# B&R Automation Studio project BottleFiller
Automation Studio 4.11.3.51 SP; technology packages: mapp 5.18.0, mappCockpit 5.18.0, mappMotion 5.18.1, mappView 5.18.1

## Configuration Config1

CPU 5PP5CP.US15-02, AutomationRuntime E4.83, Build 4.1.2, Safety 0.0, Vc V4.72.5

CPU X20CP1586, AutomationRuntime B4.92, Build 4.1.2, Vc V4.72.5

### Task classes (Cpu.sw)
```
Cyclic#4:
  RobVis <- Simulation.Logic.RobVis.prg [disabled]
  BootleFill <- BootleFiller.prg
Libraries: McBase, CoTrace, AsZip, FileIO, runtime, MpUserX, MpBase
```

### Task classes (Cpu.sw)
```
Cyclic#4:
  RobVis <- s.Logic.RobVis.prg
```

### Hardware
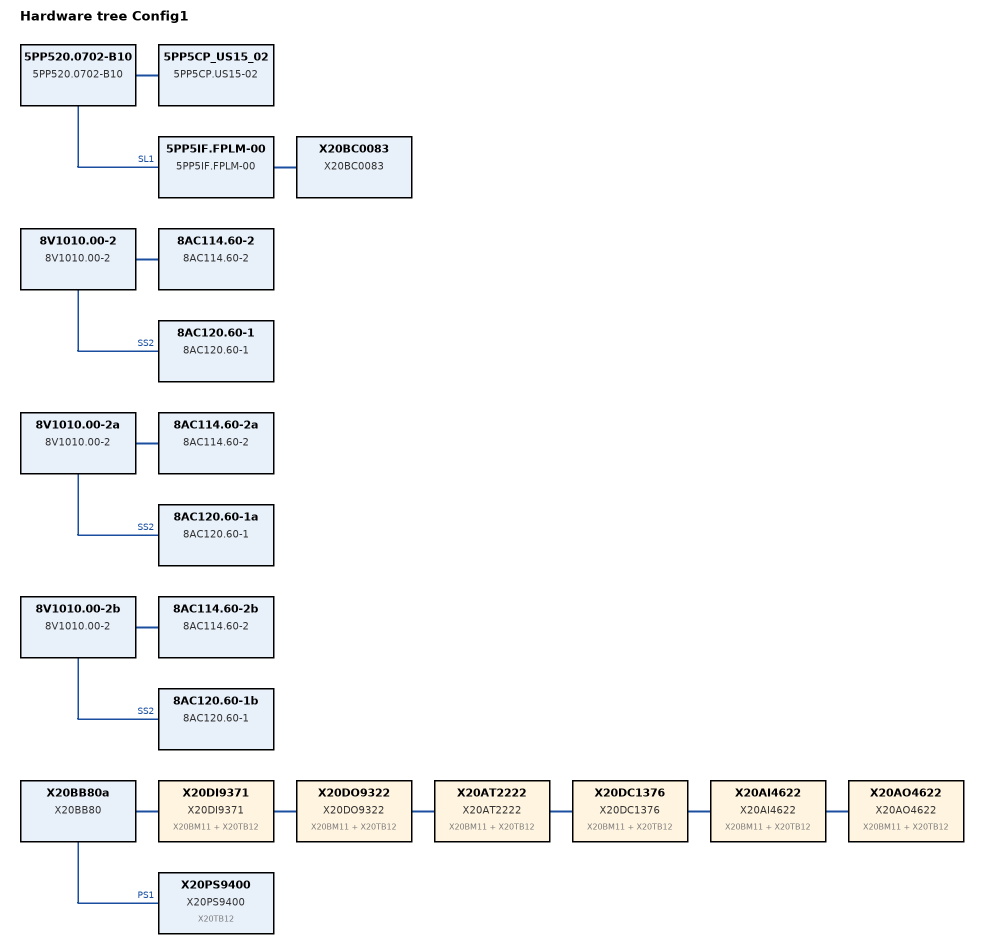
```
5PP520.0702-B10 : 5PP520.0702-B10 v2.0.1.1
  Connector IF3:
    ActivateDevice = 1
    Mode = Manual
    InternetAddress = 192.168.0.121
    SubnetMask = 255.255.255.0
    ActivateSnmp = 2
5PP5CP_US15_02 : 5PP5CP.US15-02 v2.1.6.0  [SY -> 5PP520.0702-B10.SY1]
  ConfigurationID = BottleFiller_Config1
  UserPartitionSize = 10
  FileDevice1
  FileDeviceName1 = USER
  FileDevicePath1 = C:\Recipe\
  ActivateOpcUa = 1
  OpcUaInformationModels_PV_Version = 1
5PP5IF.FPLM-00 : 5PP5IF.FPLM-00 v2.5.0.0  [SL -> 5PP520.0702-B10.SL1]
  Connector IF1:
    Channel1
    ChannelID1 = McAcpBroadcast
8AC114.60-2 : 8AC114.60-2 v1.0.0.8  [SS -> 8V1010.00-2.SS1; PLK1 -> X20BC0083.PLK2 (NodeNumber=2) [Cable Type=PowerlinkCable, Length=10, Version=1.0.0.3]; PLK2 -> 8AC114.60-2a.PLK1 (NodeNumber=2) [Cable Type=PowerlinkCable, Length=10, Version=1.0.0.3]]
8AC114.60-2a : 8AC114.60-2 v1.0.0.8  [SS -> 8V1010.00-2a.SS1; PLK1 -> 8AC114.60-2.PLK2 (NodeNumber=3) [Cable Type=PowerlinkCable, Length=10, Version=1.0.0.3]; PLK2 -> 8AC114.60-2b.PLK1 (NodeNumber=3) [Cable Type=PowerlinkCable, Length=10, Version=1.0.0.3]]
8AC114.60-2b : 8AC114.60-2 v1.0.0.8  [SS -> 8V1010.00-2b.SS1; PLK1 -> 8AC114.60-2a.PLK2 (NodeNumber=4) [Cable Type=PowerlinkCable, Length=10, Version=1.0.0.3]]
8AC120.60-1 : 8AC120.60-1 v2.2.0.0  [SS -> 8V1010.00-2.SS2]
  PlugInType = Encoder
  McAcoposTypeID = AcoposPlugInConfig
8AC120.60-1a : 8AC120.60-1 v2.2.0.0  [SS -> 8V1010.00-2a.SS2]
  PlugInType = Encoder
  McAcoposTypeID = AcoposPlugInConfig
8AC120.60-1b : 8AC120.60-1 v2.2.0.0  [SS -> 8V1010.00-2b.SS2]
  PlugInType = Encoder
  McAcoposTypeID = AcoposPlugInConfig
8V1010.00-2 : 8V1010.00-2 v2.2.0.0
  DriveConfiguration/Module:
    McAcoposTypeID = AcoposConfig
    ActivateACOPOSSimulationOnPLC = 0
    PowerSupply = ETA
  DriveConfiguration/Channel[1]/RealAxis:
    AxisReference = axisConv
    MechanicalElementsIsInvisible = 0
  DriveConfiguration/Channel[1]/RealAxis/MechanicalElements/Gearbox:
    InputIsReadOnly = 0
    Input = 1
    OutputIsReadOnly = 0
    Output = 100
  DriveConfiguration/Channel[1]/RealAxis/MechanicalElements/RotaryToLinearTransformation:
    ReferenceDistanceIsReadOnly = 0
    ReferenceDistance = 1
  DriveConfiguration/Channel[1]/RealAxis/Controller:
    ModeIsReadOnly = 0
    Mode = PositionController
  DriveConfiguration/Channel[1]/RealAxis/Controller/Mode/Position:
    ProportionalGain = 50.0
    IntegrationTime = 0.0
    PredictionTime = 0.0004
    TotalDelayTime = 0.0004
  DriveConfiguration/Channel[1]/RealAxis/Controller/Mode/Speed:
    ProportionalGainIsReadOnly = 0
    ProportionalGain = 2.0
    IntegrationTimeIsReadOnly = 0
    IntegrationTime = 0.0
    FilterTimeIsReadOnly = 0
    FilterTime = 0.0
  DriveConfiguration/Channel[1]/RealAxis/Controller/Mode/LoopFilters:
    LoopFilterXIsReadOnly = 0
    LoopFilter1 = NotUsed
    LoopFilter2 = NotUsed
    LoopFilter3 = NotUsed
  DriveConfiguration/Channel[1]/RealAxis/Homing:
    ModeIsReadOnly = 0
    Mode = Direct
  DriveConfiguration/Channel[1]/RealAxis/Homing/Mode:
    Position = 0.0
    ReferencePulse = NotUsed
  DriveConfiguration/Channel[1]/RealAxis/Homing:
    RestorePositionVariable = 
  DriveConfiguration/Channel[1]/RealAxis/StopReaction:
    QuickstopIsReadOnly = 0
    Quickstop = DecelerationLimit
    DriveErrorIsReadOnly = 0
    DriveError = DecelerationLimit
  DriveConfiguration/Channel[1]/RealAxis/MovementErrorLimits:
    PositionError = 100
    VelocityErrorMonitoring = NotUsed
  DriveConfiguration/Channel[1]/RealAxis:
    JerkFilterIsReadOnly = 0
    JerkFilter = NotUsed
  DriveConfiguration/Channel[1]/RealAxis/DigitalInputs/HomingSwitch:
    SourceIsReadOnly = 0
    Source = X1Ref
    Level = High
  DriveConfiguration/Channel[1]/RealAxis/DigitalInputs/PositiveLimitSwitch:
    Source = X1PosLim
    Level = High
  DriveConfiguration/Channel[1]/RealAxis/DigitalInputs/NegativeLimitSwitch:
    Source = X1NegLim
    Level = High
  DriveConfiguration/Channel[1]/RealAxis/DigitalInputs/Trigger1:
    Source = X1Trigger1
    Level = High
  DriveConfiguration/Channel[1]/RealAxis/DigitalInputs/Trigger2:
    Source = X1Trigger2
    Level = High
  DriveConfiguration/Channel[1]/RealAxis/DigitalInputs/Quickstop:
    Input = Trigger2
  DriveConfiguration/Channel[1]/RealAxis/Simulation:
    SimulationModeOnPLC = SetValueGeneration
    SimulationModeOnACOPOS = NotUsed
  DriveConfiguration/Channel[1]:
    ExternalEncoderAxis = NotUsed
8V1010.00-2a : 8V1010.00-2 v2.2.0.0
  DriveConfiguration/Module:
    McAcoposTypeID = AcoposConfig
    ActivateACOPOSSimulationOnPLC = 1
    PowerSupply = ETA
  DriveConfiguration/Channel[1]/RealAxis:
    AxisReference = axisCart
    MechanicalElementsIsInvisible = 0
  DriveConfiguration/Channel[1]/RealAxis/MechanicalElements/Gearbox:
    InputIsReadOnly = 0
    Input = 1
    OutputIsReadOnly = 0
    Output = 1
  DriveConfiguration/Channel[1]/RealAxis/MechanicalElements/RotaryToLinearTransformation:
    ReferenceDistanceIsReadOnly = 0
    ReferenceDistance = 1
  DriveConfiguration/Channel[1]/RealAxis/Controller:
    ModeIsReadOnly = 0
    Mode = PositionController
  DriveConfiguration/Channel[1]/RealAxis/Controller/Mode/Position:
    ProportionalGain = 50.0
    IntegrationTime = 0.0
    PredictionTime = 0.0004
    TotalDelayTime = 0.0004
  DriveConfiguration/Channel[1]/RealAxis/Controller/Mode/Speed:
    ProportionalGainIsReadOnly = 0
    ProportionalGain = 2.0
    IntegrationTimeIsReadOnly = 0
    IntegrationTime = 0.0
    FilterTimeIsReadOnly = 0
    FilterTime = 0.0
  DriveConfiguration/Channel[1]/RealAxis/Controller/Mode/LoopFilters:
    LoopFilterXIsReadOnly = 0
    LoopFilter1 = NotUsed
    LoopFilter2 = NotUsed
    LoopFilter3 = NotUsed
  DriveConfiguration/Channel[1]/RealAxis/Homing:
    ModeIsReadOnly = 0
    Mode = Direct
  DriveConfiguration/Channel[1]/RealAxis/Homing/Mode:
    Position = 0.0
    ReferencePulse = NotUsed
  DriveConfiguration/Channel[1]/RealAxis/Homing:
    RestorePositionVariable = 
  DriveConfiguration/Channel[1]/RealAxis/StopReaction:
    QuickstopIsReadOnly = 0
    Quickstop = DecelerationLimit
    DriveErrorIsReadOnly = 0
    DriveError = DecelerationLimit
  DriveConfiguration/Channel[1]/RealAxis/MovementErrorLimits:
    PositionError = 1.0
    VelocityErrorMonitoring = Automatic1
  DriveConfiguration/Channel[1]/RealAxis:
    JerkFilterIsReadOnly = 0
    JerkFilter = NotUsed
  DriveConfiguration/Channel[1]/RealAxis/DigitalInputs/HomingSwitch:
    SourceIsReadOnly = 0
    Source = X1Ref
    Level = High
  DriveConfiguration/Channel[1]/RealAxis/DigitalInputs/PositiveLimitSwitch:
    Source = X1PosLim
    Level = High
  DriveConfiguration/Channel[1]/RealAxis/DigitalInputs/NegativeLimitSwitch:
    Source = X1NegLim
    Level = High
  DriveConfiguration/Channel[1]/RealAxis/DigitalInputs/Trigger1:
    Source = X1Trigger1
    Level = High
  DriveConfiguration/Channel[1]/RealAxis/DigitalInputs/Trigger2:
    Source = X1Trigger2
    Level = High
  DriveConfiguration/Channel[1]/RealAxis/DigitalInputs/Quickstop:
    Input = Trigger2
  DriveConfiguration/Channel[1]/RealAxis/Simulation:
    SimulationModeOnPLC = SetValueGeneration
    SimulationModeOnACOPOS = CompleteControlledSystem
  DriveConfiguration/Channel[1]/RealAxis/Simulation/SimulationModeOnACOPOS:
    LoadModel = OneMassBasedOnMotorParameters
  DriveConfiguration/Channel[1]/RealAxis/Simulation/SimulationModeOnACOPOS/LoadModel:
    AdditiveLoadParID = 0
  DriveConfiguration/Channel[1]/RealAxis/AxisFeatures:
    FeatureRef[1] = Feature_CamAutomat
  DriveConfiguration/Channel[1]:
    ExternalEncoderAxis = NotUsed
8V1010.00-2b : 8V1010.00-2 v2.2.0.0
  DriveConfiguration/Module:
    McAcoposTypeID = AcoposConfig
    ActivateACOPOSSimulationOnPLC = 1
    PowerSupply = ETA
  DriveConfiguration/Channel[1]/RealAxis:
    AxisReference = axisNozzle
    MechanicalElementsIsInvisible = 0
  DriveConfiguration/Channel[1]/RealAxis/MechanicalElements/Gearbox:
    InputIsReadOnly = 0
    Input = 1
    OutputIsReadOnly = 0
    Output = 1
  DriveConfiguration/Channel[1]/RealAxis/MechanicalElements/RotaryToLinearTransformation:
    ReferenceDistanceIsReadOnly = 0
    ReferenceDistance = 1
  DriveConfiguration/Channel[1]/RealAxis/Controller:
    ModeIsReadOnly = 0
    Mode = PositionController
  DriveConfiguration/Channel[1]/RealAxis/Controller/Mode/Position:
    ProportionalGain = 2
    IntegrationTime = 0.0
    PredictionTime = 0.0004
    TotalDelayTime = 0.0004
  DriveConfiguration/Channel[1]/RealAxis/Controller/Mode/Speed:
    ProportionalGainIsReadOnly = 0
    ProportionalGain = 0.01
    IntegrationTimeIsReadOnly = 0
    IntegrationTime = 0.0
    FilterTimeIsReadOnly = 0
    FilterTime = 0.0
  DriveConfiguration/Channel[1]/RealAxis/Controller/Mode/LoopFilters:
    LoopFilterXIsReadOnly = 0
    LoopFilter1 = NotUsed
    LoopFilter2 = NotUsed
    LoopFilter3 = NotUsed
  DriveConfiguration/Channel[1]/RealAxis/Homing:
    ModeIsReadOnly = 0
    Mode = Direct
  DriveConfiguration/Channel[1]/RealAxis/Homing/Mode:
    Position = 195.0
    ReferencePulse = NotUsed
  DriveConfiguration/Channel[1]/RealAxis/Homing:
    RestorePositionVariable = 
  DriveConfiguration/Channel[1]/RealAxis/StopReaction:
    QuickstopIsReadOnly = 0
    Quickstop = DecelerationLimit
    DriveErrorIsReadOnly = 0
    DriveError = DecelerationLimit
  DriveConfiguration/Channel[1]/RealAxis/MovementErrorLimits:
    PositionError = 1.0
    VelocityErrorMonitoring = Automatic1
  DriveConfiguration/Channel[1]/RealAxis:
    JerkFilterIsReadOnly = 0
    JerkFilter = NotUsed
  DriveConfiguration/Channel[1]/RealAxis/DigitalInputs/HomingSwitch:
    SourceIsReadOnly = 0
    Source = X1Ref
    Level = High
  DriveConfiguration/Channel[1]/RealAxis/DigitalInputs/PositiveLimitSwitch:
    Source = X1PosLim
    Level = High
  DriveConfiguration/Channel[1]/RealAxis/DigitalInputs/NegativeLimitSwitch:
    Source = X1NegLim
    Level = High
  DriveConfiguration/Channel[1]/RealAxis/DigitalInputs/Trigger1:
    Source = X1Trigger1
    Level = High
  DriveConfiguration/Channel[1]/RealAxis/DigitalInputs/Trigger2:
    Source = X1Trigger2
    Level = High
  DriveConfiguration/Channel[1]/RealAxis/DigitalInputs/Quickstop:
    Input = Trigger2
  DriveConfiguration/Channel[1]/RealAxis/Simulation:
    SimulationModeOnPLC = SetValueGeneration
    SimulationModeOnACOPOS = NotUsed
  DriveConfiguration/Channel[1]/RealAxis/AxisFeatures:
    FeatureRef[1] = Feature_CamList
  DriveConfiguration/Channel[1]:
    ExternalEncoderAxis = NotUsed
  DriveConfiguration/Channel[1]/ChannelFeatures:
    FeatureRef[1] = Feature_CamList_1
X20AI4622 : X20AI4622 v1.2.0.0  [SS1 -> X20TB12f.SS; SL -> X20BM11e.SL1]
X20AO4622 : X20AO4622 v1.3.0.0  [SS1 -> X20TB12g.SS; SL -> X20BM11f.SL1]
X20AT2222 : X20AT2222 v1.4.0.0  [SS1 -> X20TB12d.SS; SL -> X20BM11c.SL1]
X20BB80a : X20BB80 v1.1.0.0
X20BC0083 : X20BC0083 v2.12.0.0  [PLK1 -> 5PP5IF.FPLM-00.IF1 (NodeNumber=1) [Cable Type=PowerlinkCable, Length=10, Version=1.0.0.3]; PLK2 -> 8AC114.60-2.PLK1 (NodeNumber=1) [Cable Type=PowerlinkCable, Length=10, Version=1.0.0.3]; SL -> X20BB80a.SL1]
  Supervision = off
X20BM11a : X20BM11 v1.1.0.0  [X2X1 -> X20BB80a.IF1]
X20BM11b : X20BM11 v1.1.0.0  [X2X1 -> X20BM11a.X2X2]
X20BM11c : X20BM11 v1.1.0.0  [X2X1 -> X20BM11b.X2X2]
X20BM11d : X20BM11 v1.1.0.0  [X2X1 -> X20BM11c.X2X2]
X20BM11e : X20BM11 v1.1.0.0  [X2X1 -> X20BM11d.X2X2]
X20BM11f : X20BM11 v1.1.0.0  [X2X1 -> X20BM11e.X2X2]
X20DC1376 : X20DC1376 v1.3.0.0  [SS1 -> X20TB12e.SS; SL -> X20BM11d.SL1]
X20DI9371 : X20DI9371 v1.3.0.0  [SS1 -> X20TB12a.SS; SL -> X20BM11a.SL1]
X20DO9322 : X20DO9322 v1.4.0.0  [SS1 -> X20TB12c.SS; SL -> X20BM11b.SL1]
X20PS9400 : X20PS9400 v1.7.0.0  [SS1 -> X20TB12b.SS; PS -> X20BB80a.PS1]
  Supervision = off
X20TB12a : X20TB12 v1.0.0.0
X20TB12b : X20TB12 v1.0.0.0
X20TB12c : X20TB12 v1.0.0.0
X20TB12d : X20TB12 v1.0.0.0
X20TB12e : X20TB12 v1.0.0.0
X20TB12f : X20TB12 v1.0.0.0
X20TB12g : X20TB12 v1.0.0.0
```

### Config_1.axis - 5PP5CP_US15_02/mappMotion/Config_1.axis
```
Element axisConv (Type=axis)
  BaseTypeIsReadOnly = 0
  BaseType = LinearPeriodic
    MeasurementUnit = 5066068
    MeasurementResolutionIsReadOnly = 0
    MeasurementResolution = 0.01
    CountDirectionIsReadOnly = 0
    CountDirection = Standard
    PeriodSettings:
      Period = 5000
  MovementLimitsIsReadOnly = 0
  MovementLimits = Internal
    Position:
      LowerLimitMin = -1.79769313486231E308
      UpperLimitMax = 1.79769313486231E308
      LowerLimit = -1000.0
      UpperLimit = 1000.0
    VelocityIsReadOnly = 0
    Velocity:
      VelocityMax = 3.4E38
      Velocity = 10.0
    AccelerationIsReadOnly = 0
    Acceleration:
      AccelerationMax = 3.4E38
      Acceleration = 50.0
    DecelerationIsReadOnly = 0
    Deceleration:
      DecelerationMax = 3.4E38
      Deceleration = 50.0
  Alarms = None
Element axisCart (Type=axis)
  BaseTypeIsReadOnly = 0
  BaseType = LinearPeriodic
    MeasurementUnit = 5066068
    MeasurementResolutionIsReadOnly = 0
    MeasurementResolution = 0.01
    CountDirectionIsReadOnly = 0
    CountDirection = Standard
    PeriodSettings:
      Period = 1200
  MovementLimitsIsReadOnly = 0
  MovementLimits = Internal
    Position:
      LowerLimitMin = -1.79769313486231E308
      UpperLimitMax = 1.79769313486231E308
      LowerLimit = -1000.0
      UpperLimit = 1000.0
    VelocityIsReadOnly = 0
    Velocity:
      VelocityMax = 3.4E38
      Velocity = 10.0
    AccelerationIsReadOnly = 0
    Acceleration:
      AccelerationMax = 3.4E38
      Acceleration = 50.0
    DecelerationIsReadOnly = 0
    Deceleration:
      DecelerationMax = 3.4E38
      Deceleration = 50.0
  Alarms = None
Element axisNozzle (Type=axis)
  BaseTypeIsReadOnly = 0
  BaseType = LinearPeriodic
    MeasurementUnit = 5066068
    MeasurementResolutionIsReadOnly = 0
    MeasurementResolution = 0.01
    CountDirectionIsReadOnly = 0
    CountDirection = Standard
    PeriodSettings:
      Period = 200
  MovementLimitsIsReadOnly = 0
  MovementLimits = Internal
    Position:
      LowerLimitMin = -1.79769313486231E308
      UpperLimitMax = 1.79769313486231E308
      LowerLimit = -1000.0
      UpperLimit = 1000.0
    VelocityIsReadOnly = 0
    Velocity:
      VelocityMax = 3.4E38
      Velocity = 10.0
    AccelerationIsReadOnly = 0
    Acceleration:
      AccelerationMax = 3.4E38
      Acceleration = 50.0
    DecelerationIsReadOnly = 0
    Deceleration:
      DecelerationMax = 3.4E38
      Deceleration = 50.0
  Alarms = None
```

### Config_1.camlist - 5PP5CP_US15_02/mappMotion/Config_1.camlist
```
Element CamList_1 (Type=camlist)
  Row[1]:
    CamName = b1_Nozzle
    CamID = 1
    Description
```

### Config_2.axisfeature - 5PP5CP_US15_02/mappMotion/Config_2.axisfeature
```
Element Feature_CamList_1 (Type=axisfeature)
  Type = CamList
    CamListRef = CamList_1
```

### configAxis.axis - 5PP5CP_US15_02/mappMotion/configAxis.axis
```
Element axisConv (Type=axis)
  BaseTypeIsReadOnly = 0
  BaseType = LinearPeriodic
    MeasurementUnit = 5066068
    MeasurementResolutionIsReadOnly = 0
    MeasurementResolution = 0.01
    CountDirectionIsReadOnly = 0
    CountDirection = Standard
    PeriodSettings:
      Period = 5000
  MovementLimitsIsReadOnly = 0
  MovementLimits = Internal
    Position:
      LowerLimitMin = -1.79769313486231E308
      UpperLimitMax = 1.79769313486231E308
      LowerLimit = -1000.0
      UpperLimit = 1000.0
    VelocityIsReadOnly = 0
    Velocity:
      VelocityMax = 3.4E38
      Velocity = 600
    AccelerationIsReadOnly = 0
    Acceleration:
      AccelerationMax = 3.4E38
      Acceleration = 10000
    DecelerationIsReadOnly = 0
    Deceleration:
      DecelerationMax = 3.4E38
      Deceleration = 100000
  Alarms = MpAlarmX
    mapp.AlarmX.Core.Configuration:
      [0]:
        Message = Conveyor system problem
        Code = 100
        Severity = 10
      [3]:
        Message = Conveyor Operation Problem
        Code = 200
        Severity = 20
      [14]:
        Message = Conveyor Motor problem
        Code = 300
        Severity = 30
Element axisCart (Type=axis)
  BaseTypeIsReadOnly = 0
  BaseType = LinearBounded
    MeasurementUnit = 5066068
    MeasurementResolutionIsReadOnly = 0
    MeasurementResolution = 0.01
    CountDirectionIsReadOnly = 0
    CountDirection = Standard
  MovementLimitsIsReadOnly = 0
  MovementLimits = Internal
    Position:
      LowerLimitMin = -1.79769313486231E308
      UpperLimitMax = 1.79769313486231E308
      LowerLimit = -100
      UpperLimit = 1100
    VelocityIsReadOnly = 0
    Velocity:
      VelocityMax = 3.4E38
      Velocity = 800
    AccelerationIsReadOnly = 0
    Acceleration:
      AccelerationMax = 3.4E38
      Acceleration = 10000
    DecelerationIsReadOnly = 0
    Deceleration:
      DecelerationMax = 3.4E38
      Deceleration = 100000
  Alarms = MpAlarmX
    mapp.AlarmX.Core.Configuration:
      [0]:
        Message = Cart System problem
        Code = 101
        Severity = 10
      [3]:
        Message = Cart Operation problem
        Code = 201
        Severity = 20
      [14]:
        Message = Cart Motor problem
        Code = 301
        Severity = 30
Element axisNozzle (Type=axis)
  BaseTypeIsReadOnly = 0
  BaseType = LinearBounded
    MeasurementUnit = 5066068
    MeasurementResolutionIsReadOnly = 0
    MeasurementResolution = 0.01
    CountDirectionIsReadOnly = 0
    CountDirection = Standard
  MovementLimitsIsReadOnly = 0
  MovementLimits = Internal
    Position:
      LowerLimitMin = -1.79769313486231E308
      UpperLimitMax = 1.79769313486231E308
      LowerLimit = 0
      UpperLimit = 200
    VelocityIsReadOnly = 0
    Velocity:
      VelocityMax = 3.4E38
      Velocity = 5000
    AccelerationIsReadOnly = 0
    Acceleration:
      AccelerationMax = 3.4E38
      Acceleration = 20000
    DecelerationIsReadOnly = 0
    Deceleration:
      DecelerationMax = 3.4E38
      Deceleration = 800000
  Alarms = MpAlarmX
    mapp.AlarmX.Core.Configuration:
      [0]:
        Message = Nozzle System problem
        Code = 102
        Severity = 10
      [3]:
        Message = Nozzle Operation problem
        Code = 202
        Severity = 20
      [14]:
        Message = Nozzle Motor problem
        Code = 302
        Severity = 30
```

### configCam.axisfeature - 5PP5CP_US15_02/mappMotion/configCam.axisfeature
```
Element Feature_CamAutomat (Type=axisfeature)
  Type = CamAutomat
    CamAutomatType = ACOPOS
      CommonParameters:
        Master:
          ValueSource = SetPosition
            AxisReference
            MaxVelocity = 1.0
          StartPosition = 0.0
          StartInterval = MasterAxisPeriod
        AdvancedParameters:
          StartStateParameters:
            StartState = 0
            RelMasterStartPos = 0.0
          AdditiveAxes:
            AdditiveMasterValueSource = NotUsed
            AdditiveSlaveValueSource = NotUsed
          MasterStartPositionMode = NotEvaluatedAnew
          ControlSettings:
            CrossLeftBoundary = PositionLimitedHorizontal
            CamChangeImmediately = CurrentMasterMoveDir
          MessageSettings:
            ErrorsInStandby = NoErrorMessages
          TriggerAndLatch:
            Trigger1Delay = 0.0
            Trigger2Delay = 0.0
            SlaveLatchParID = 0
          EventParIDs
          StartIntervals
          Factors:
            SlaveFactorParID = 0
      States:
        State0 = Used
```

### configNozz.axisfeature - 5PP5CP_US15_02/mappMotion/configNozz.axisfeature
```
Element Feature_CamList (Type=axisfeature)
  Type = CamAutomat
    CamAutomatType = ACOPOS
      CommonParameters:
        Master:
          ValueSource = SetPosition
            AxisReference = axisConv
            MaxVelocity = 600
          StartPosition = 0.0
          StartInterval = MasterAxisPeriod
        AdvancedParameters:
          StartStateParameters:
            StartState = 0
            RelMasterStartPos = 0.0
          AdditiveAxes:
            AdditiveMasterValueSource = NotUsed
            AdditiveSlaveValueSource = NotUsed
          MasterStartPositionMode = NotEvaluatedAnew
          ControlSettings:
            CrossLeftBoundary = PositionLimitedHorizontal
            CamChangeImmediately = CurrentMasterMoveDir
          MessageSettings:
            ErrorsInStandby = NoErrorMessages
          TriggerAndLatch:
            Trigger1Delay = 0.0
            Trigger2Delay = 0.0
            SlaveLatchParID = 0
          EventParIDs
          StartIntervals
          Factors:
            SlaveFactorParID = 0
      States:
        State0 = Used
          Events:
            Event[0]:
              Type = Signal1FromPLC
              Transition = Immediately
              SynchronousUpdate = Used
              NextState = 1
        State[1]:
          Cam = Predefined
            PredefinedCam = ZeroPoint
          MasterFactor = 100
          SlaveFactor = -100
          CompensationMode = MasterSlaveAbsolutePosition
            MasterPosition = 90
            SlavePosition = 195
            MaxSlaveVelocity = 1000
            MaxSlaveAcceleration1 = 2000
            MaxSlaveAcceleration2 = 2250
            AdvancedParameters = NotUsed
          AdvancedParameters:
            RepeatCounterInit = 0
            MasterValueSource = CommonMaster
          Events:
            Event[0]:
              Type = StateEnd
              Transition = EndOfState
              SynchronousUpdate = NotUsed
              NextState = 2
        State[2]:
          Cam = Predefined
            PredefinedCam = OneToOne
          MasterFactor = 100
          SlaveFactor = 100
          CompensationMode = SlaveCompensationAbsSlPos
            MasterDistance = 50
            SlavePosition = 5
            AdvancedParameters = NotUsed
          AdvancedParameters:
            RepeatCounterInit = 0
            MasterValueSource = CommonMaster
          Events:
            Event[0]:
              Type = StateEnd
              Transition = EndOfState
              SynchronousUpdate = NotUsed
              NextState = 3
        State[3]:
          Cam = CamID
            CamID = 1
          MasterFactor = 40000
          SlaveFactor = 19000
          CompensationMode = NoCompensation
          AdvancedParameters:
            RepeatCounterInit = 0
            MasterValueSource = CommonMaster
          Events:
            Event[0]:
              Type = StateEnd
              Transition = EndOfState
              SynchronousUpdate = NotUsed
              NextState = 4
        State[4]:
          Cam = Predefined
            PredefinedCam = ZeroPoint
          MasterFactor = 100
          SlaveFactor = 100
          CompensationMode = SlaveCompensationAbsSlPos
            MasterDistance = 50
            SlavePosition = 195
            AdvancedParameters = NotUsed
          AdvancedParameters:
            RepeatCounterInit = 0
            MasterValueSource = CommonMaster
          Events:
            Event[0]:
              Type = StateEnd
              Transition = Immediately
              SynchronousUpdate = NotUsed
              NextState = 2
```

### alarm.mpalarmxcore - 5PP5CP_US15_02/mappServices/alarm.mpalarmxcore
```
Element gBFAlarmXCore (Type=mpalarmxcore)
  mapp.AlarmX.Core.Configuration:
    [0]:
      Name = noPower
      Message = You should click PowerSwitch first.
      Code = 99
      Severity = 10
      Behavior = PersistentAlarm
```

### fileM.mpfilemanager - 5PP5CP_US15_02/mappServices/fileM.mpfilemanager
```
Element FileManagement (Type=mpfilemanager)
  FileManager:
    Devices:
      0:
        DeviceName = USER
        Text = Recipe
    Access:
      0:
        Folder = *
        Roles:
          0:
            Role = Shift Leader
            Rights:
              Visible = TRUE
              FolderRead = TRUE
              FileRead = TRUE
              FileEdit = TRUE
              FolderEdit = TRUE
    Auditing = MpAudit
      Read = TRUE
  FileManagerRestrict:
    0:
      0:
        Folder = 
    1:
      Functionality = TextEditor
      0:
        Folder = C:\Recipe
        Restrictions:
          BrowseUp = TRUE
          BrowseDown = TRUE
          ReadOnly = TRUE
          CreatFolders = TRUE
```

### recipeXML.mprecipexml - 5PP5CP_US15_02/mappServices/recipeXML.mprecipexml
```
Element BFRecipe (Type=mprecipexml)
  mapp.Recipe.Xml:
    Auditing = MpAudit
```

## Logical view

Binary libraries used (declarations not repeated): operator, runtime, astime, AsIecCon, McBase, CoTrace, AsZip, FileIO, MpUserX, MpBase

### Global.var - Global variables
```iecst
VAR
	roleInfo : MpUserXMgrUIRoleInfoType;
	role : MpUserXMgrUIUserInfoType;
END_VAR
```

### Package Logical/Libraries - Global libraries

### BF_GlobarVar.var
```iecst
VAR
	gFillerTyp : gBFWorkEnum;
	gAxisCase : gBFCaseEnum;
	gControl : gManagementTyp;
	gAxisUpdate : gAxisUpdateParType;
	gMainAction : gMainActionTyp;
	gAxisOutputs : gAxisOutputsTyp;
	gCamSeqParam : camSequencersParams;
	gCaseError : gErrorCaseEnum;
	gMain : gFillerEnum;
	gPump : gPumpMgmtTyp;
	temp : BOOL := FALSE;
END_VAR
```

### BF_GlobalTyp.typ
```iecst
TYPE
	gPumpMgmtTyp : 	STRUCT
		PumpFlowSpeed : USINT;
		PumpRelay : USINT := 0;
		ValveStatus : STRING[80];
		ValveRelay : BOOL := FALSE;
	END_STRUCT;
	camSequencersParams : 	STRUCT
		cart : camParam; (*Parametry cama karetki*)
		nozzle : camParam; (*Parametry cama dysz*)
	END_STRUCT;
	camParam : 	STRUCT
		signal1 : BOOL := FALSE; (*Wyzwalanie signal1*)
		currentStateIndex : INT := 0; (*Zwraca aktualny state*)
	END_STRUCT;
	gAxisOutputsTyp : 	STRUCT
		Conveyor : gControlInfoTyp;
		Cart : gControlInfoTyp;
		Nozzle : gControlInfoTyp;
		currentBottleType : UINT := 1; (*Aktualny typ butelki*)
		velocity : REAL; (*Aktualna prędkość*)
	END_STRUCT;
	gControlInfoTyp : 	STRUCT  (*parameters, output*)
		error : BOOL := FALSE; (*error*)
		isPowered : BOOL := FALSE; (*jest zasilony*)
		isHomed : BOOL := FALSE; (*jest w pozycji home*)
		position : REAL := 0; (*aktualna pozycja*)
		velocity : REAL := 0; (*aktualne velocity*)
		updateDone : BOOL := FALSE;
		MoveActive : BOOL := FALSE;
		Direction : STRING[80];
	END_STRUCT;
	gControlTyp : 	STRUCT  (*parameters, inputs*)
		power : BOOL := FALSE; (*Uruchomienie maszyny*)
		errorReset : BOOL := FALSE;
		autoTune : BOOL := TRUE;
		home : BOOL := FALSE;
		jogNegative : BOOL := FALSE;
		jogPositive : BOOL := FALSE;
		moveVelocity : BOOL := FALSE;
		stop : BOOL := FALSE;
		currentBottleType : STRING[80] := '1';
		safeLevelStop : BOOL; (*Informuje, czy w trybie półautomatycznym przekroczone zostały bezpieczne granice*)
		onlyLeft : BOOL := FALSE; (*Wskazuje, że w trybie półautomatycznym możliwy aktualnie jest ruch tylko w lewo*)
		onlyRight : BOOL := FALSE; (*Wskazuje, że w trybie półautomatycznym możliwy aktualnie jest ruch tylko w prawo*)
		upperLimit : INT; (*Maksymalne velocity Operatora*)
		lowerLimit : INT; (*Minimalne velocity Operatora*)
		Direction : STRING[80];
	END_STRUCT;
	gMainActionTyp : 	STRUCT  (*Flagi pomocne w sterowaniu projektem*)
		powered : BOOL := FALSE; (*Czy maszyna jest zasilona*)
		homed : BOOL := FALSE; (*Czy maszyna jest home'owana*)
		connected : BOOL := FALSE; (*Czy osie są połączone*)
		disconnected : BOOL := FALSE; (*Czy osie są rozłączone*)
		stopped : BOOL := FALSE; (*Czy Osie stoją*)
	END_STRUCT;
	gAxisUpdateParType : 	STRUCT  (*update parameters structure*)
		Conveyor : gParametersUpdate;
		Cart : gParametersUpdate;
		Nozzle : gParametersUpdate;
		staticVelocity : STRING[80] := '10'; (*Static velocity to veloocity z opcji "Slow", "Normal", "Fast"*)
	END_STRUCT;
	gManagementTyp : 	STRUCT  (*Zarządzanie maszyną*)
		Conveyor : gControlTyp;
		Cart : gControlTyp;
		Nozzle : gControlTyp;
		power : BOOL := FALSE; (*Zasilenie maszyny*)
		start : BOOL := FALSE; (*Start maszyny*)
		stop : BOOL := FALSE; (*Stop maszyny*)
		manual : BOOL := FALSE; (*Manualna praca*)
		inCam : BOOL := FALSE; (*Flaga wskazująca na status połączenia osi*)
		needUpdate : BOOL := TRUE; (*Flaga wskazująca na konieczność aktualizacji*)
		moveVelocity : BOOL := FALSE; (*Wyzwolenie ruchu*)
		disconnect : BOOL := FALSE; (*Rozłączenie osi*)
		bottleCnt : INT := 0; (*Liczy butelki*)
		currentBottleType : STRING[80] := '1'; (*Aktualny typ butelki*)
		part : REAL; (*5% z aktualnej prędkości*)
		partVelUpd : BOOL := FALSE; (*Flaga wskazująca na konieczność aktualizacji prędkości*)
		maxVelocity : REAL; (*Maksymalne Velocity Operatora*)
		decVisible : BOOL := TRUE; (*Widoczność przycisku Decrease*)
		emergencySTOP : BOOL := FALSE;
		switchToAutomat : BOOL := FALSE;
		incVisible : BOOL := TRUE; (*Widoczność przycisku Increase*)
		minVelocity : REAL; (*Minimalne Velocity Operatora*)
		startSeq : BOOL := TRUE;
	END_STRUCT;
	gErrorCaseEnum :
		(
		noError,
		handleError,
		inError
		);
	gFillerEnum :
		( (*Every possible case*)
		DISABLED,
		INIT,
		WORK,
		STOP,
		ERROR
		);
	gParametersUpdate : 	STRUCT  (*update parameters*)
		Velocity : REAL := 10;
		Direction : REAL := 1;
		FirstPosition : REAL := 0;
		LastPosition : REAL := 0;
		Position : REAL := 0;
		Homing : REAL := 0;
	END_STRUCT;
	gBFWorkEnum :
		( (*BF_Work control*)
		WAITING, (*Stan początkowy*)
		AUTOMAT, (*Tryb automatyczny*)
		MANUAL (*Tryb manualny*)
		);
	gBFCaseEnum :
		( (*BF_Axis control*)
		WAIT, (*Tryb początkowy*)
		STANDSTILL, (*Czeka na ruch*)
		POWERED, (*Maszyna zasilona*)
		HOLDON, (*Zatrzymanie maszyny*)
		CONNECT, (*Połączenie osi*)
		onMOVE, (*W ruchu*)
		DISCONNECT, (*Rozłączenie osi*)
		HOMING (*Przywrócenie pozycji początkowych*)
		);
END_TYPE
```

### Program Logical/BottleFiller/BF_Main (IEC)

#### Types.typ
```iecst
TYPE
	SimulationAxisPositionEnum : 	STRUCT
		Conveyor : REAL;
		Cart : REAL;
		Nozzle : REAL;
	END_STRUCT;
	bottleFillerRecipeEnum : 	STRUCT
		diPumpSpeedFlow : INT := 0;
		diVelocity : REAL := 0.0;
		diSpeedProfile : INT := 0;
		diBottleShape : INT := 0;
	END_STRUCT;
END_TYPE
```

#### Variables.var
```iecst
(*case machine*)
VAR
	bottleFillerRecipeTyp : bottleFillerRecipeEnum;
END_VAR
(*digital inputs*)
VAR
	diError : BOOL;
	diManual : BOOL := FALSE; (*Determine if machine works automatically or needs manual control*)
	diStop : BOOL := FALSE; (*Stop switch*)
	diStart : BOOL := FALSE; (*Start switch*)
	diPowerSwitch : BOOL := FALSE; (*Power on switch*)
	diLiquidLevel : REAL := 100;
	diConveyorHomingSwitch : BOOL := FALSE; (*Sensor detecting conveyor at homing position*)
	diNozzleHomingSwitch : BOOL := FALSE; (*Sensor detecting nozzle at homing position*)
	diCartHomingSwitch : BOOL := FALSE; (*Sensor detecting cart at homing position*)
	diBottleDetection : BOOL := FALSE; (*Sensor detecting presence of a bottle*)
END_VAR
(*digital outputs*)
VAR
	doPumpRelay : INT; (*Output controlling the pump building pressure for liquid flow*)
	doValveRelay : BOOL; (*Output controlling the liquid valve opening*)
END_VAR
(*analog outputs*)
VAR
	aoPumpFlowSpeed : ARRAY[0..100] OF INT; (*Datapoint in percentage to the pump system about liquid flow speed in percent*)
END_VAR
(*other variables*)
VAR
	result : INT;
	counter : INT;
	roleInfo : MpUserXMgrUIRoleInfoType;
	MpBFRecipeXml : MpRecipeXml;
	MpBFRecipeRegPar : MpRecipeRegPar; (*MpBFRecipeHMI : MpRecipeUI;
	UISetup : MpRecipeUISetupType;
	MpRecipeUIConnectType : MpRecipeUIConnectType;*)
	inCam : BOOL;
	SimulationAxisPosition : SimulationAxisPositionEnum;
	changedPosition : BOOL;
END_VAR
```

#### Main.st
```iecst
PROGRAM _INIT
	(* Insert code here *)
	 gMain:=DISABLED;
END_PROGRAM

PROGRAM _CYCLIC
	(* Insert code here *)

	SimulationAxisPosition.Cart := LREAL_TO_REAL(gAxisOutputs.Cart.position);
	SimulationAxisPosition.Conveyor := LREAL_TO_REAL(gAxisOutputs.Conveyor.position);
	SimulationAxisPosition.Nozzle := LREAL_TO_REAL(gAxisOutputs.Nozzle.position);
	gAdrAxesPositions := ADR(SimulationAxisPosition);

	CASE gMain OF
		DISABLED:
			diStart:=0;
			diStop:=0;

			IF gControl.power THEN
				gMain:=INIT;
			END_IF;

		INIT:
			gControl.Cart.lowerLimit:=-95;
			gControl.Cart.upperLimit:=1095;

			gControl.Conveyor.lowerLimit:=0;
			gControl.Conveyor.upperLimit:=4997;

			gControl.Nozzle.lowerLimit:=2;
			gControl.Nozzle.upperLimit:=197;

			gAxisCase:=POWERED;

			IF gMainAction.powered AND NOT gControl.inCam THEN
				gAxisCase:=HOMING;
			END_IF;

			IF gMainAction.powered AND gMainAction.homed THEN
				gControl.Cart.home:=0;
				gControl.Conveyor.home:=0;
				gControl.Nozzle.home:=0;
				gAxisCase:=STANDSTILL;
			END_IF;

			IF gMainAction.powered AND gMainAction.homed AND gControl.start AND NOT gControl.manual THEN
				gAxisCase:=CONNECT;
				IF gMainAction.connected THEN
					gAxisCase:=onMOVE;
					gFillerTyp:=AUTOMAT;
					gMain:=WORK;
				END_IF;
			END_IF;

			IF gMainAction.powered AND gMainAction.homed AND gControl.start AND gControl.manual THEN
				gMainAction.homed:=0;
				gAxisCase:=onMOVE;
				gFillerTyp:=MANUAL;
				gMain:=WORK;
			END_IF;

		WORK:
			result:= gControl.bottleCnt MOD 5;

			IF result=1 THEN
				gCamSeqParam.nozzle.signal1:=1;
			END_IF;
			IF result <> 1 THEN
				gCamSeqParam.nozzle.signal1:=0;
				gCamSeqParam.cart.signal1:=0;
			END_IF;

			IF (gCamSeqParam.nozzle.currentStateIndex = 3) AND (gAxisOutputs.Nozzle.position > 0 AND gAxisOutputs.Nozzle.position < 170) THEN
				gPump.ValveRelay:=1;
				gPump.ValveStatus:='Opened';
			ELSE
				gPump.ValveRelay:=0;
				gPump.ValveStatus:='Closed';
			END_IF;

		ERROR:

			IF EDGENEG(gControl.emergencySTOP) THEN
				gMain:=WORK;
			END_IF;

		STOP:

	END_CASE;

END_PROGRAM

PROGRAM _EXIT
	(* Insert code here *)

END_PROGRAM
```

### GlobalRobVis.typ - Global data types
```iecst
TYPE
	AxesPositionsType : 	STRUCT
		Conveyor : REAL;
		Cart : REAL;
		Nozzle : REAL;
	END_STRUCT;
	MachineDigitalInputsType : 	STRUCT
		BottleDetecttion : BOOL;
		ConveyorHomingSwitch : BOOL;
		CartHomingSwitch : BOOL;
		NozzleHomingSwitch : BOOL;
	END_STRUCT;
	MachineAPIType : 	STRUCT
		DigitalInputs : MachineDigitalInputsType;
	END_STRUCT;
END_TYPE
```

### Program Logical/BottleFiller/workTasks/BF_Work (IEC)

#### Variables.var
```iecst
VAR
	tempVelocity : REAL;
	switch : INT := 0;
END_VAR
```

#### Main.st
```iecst
PROGRAM _INIT
	(* Insert code here *)
END_PROGRAM

PROGRAM _CYCLIC
	(* Insert code here *)

	CASE gFillerTyp OF

		MANUAL:
			//wyłączenie jegów od razu po zatrzymaniu ruchu - wcześniej był błąd
			IF EDGENEG(gAxisOutputs.Cart.MoveActive) THEN
				gControl.Cart.jogNegative:=0;
				gControl.Cart.jogPositive:=0;
			END_IF;

			IF EDGENEG(gAxisOutputs.Conveyor.MoveActive) THEN
				gControl.Conveyor.jogNegative:=0;
				gControl.Conveyor.jogPositive:=0;
			END_IF;
			IF 	EDGENEG(gAxisOutputs.Nozzle.MoveActive) THEN
				gControl.Nozzle.jogNegative:=0;
				gControl.Nozzle.jogPositive:=0;
			END_IF;

			//Switch zależny od tego, czy osie mają być połączone, czy rozłączone
			IF EDGEPOS(gControl.inCam) THEN
				switch:=1;
			END_IF;

			IF EDGENEG(gControl.inCam) THEN
				switch:=2;
			END_IF;

			//łączenie osi
			IF switch=1 OR EDGEPOS(gControl.inCam) THEN
				IF NOT gMainAction.stopped THEN
					gAxisCase:=HOLDON;
				END_IF;

				IF gMainAction.stopped AND NOT gMainAction.homed THEN
					gAxisCase:=HOMING;
				END_IF;

				IF gMainAction.stopped AND gMainAction.homed AND NOT gMainAction.connected THEN
					gControl.Cart.home:=0;
					gControl.Conveyor.home:=0;
					gControl.Nozzle.home:=0;
					gControl.startSeq:=1;
					gMainAction.disconnected:=0;
					gAxisCase:=CONNECT;
				END_IF;

				IF gMainAction.stopped AND gMainAction.connected AND gMainAction.homed THEN
					gMainAction.homed:=0;
					gMainAction.stopped:=0;
					gAxisCase:=onMOVE;
					switch:=3;
				END_IF;
			END_IF;

			//rozłączanie osi
			IF switch=2 OR EDGENEG(gControl.inCam) THEN
				IF NOT gMainAction.disconnected THEN
					gAxisCase:=DISCONNECT;
					gMainAction.connected:=0;
				END_IF;

				IF gMainAction.disconnected THEN
					gControl.Cart.home:=0;
					gControl.Conveyor.home:=0;
					gControl.Nozzle.home:=0;
					gMainAction.homed:=0;
					gAxisCase:=onMOVE;
					IF gAxisCase=onMOVE THEN
						switch:=4;
					END_IF;
				END_IF;
			END_IF;

			//wchodzenie ponownie w tryb automatyczny
			IF NOT gControl.manual AND NOT temp THEN
				gControl.switchToAutomat:=1;
				IF NOT gMainAction.stopped THEN
					gAxisCase:=HOLDON;
				END_IF;

				gAxisUpdate.Conveyor.Velocity:=tempVelocity;
				gControl.needUpdate:=1;

				IF gMainAction.stopped AND switch=4 THEN
					gAxisCase:=HOMING;
				END_IF;

				IF (switch=3 AND gMainAction.stopped) OR (switch=4 AND gMainAction.homed) THEN
					gAxisCase:=CONNECT;
					gMainAction.disconnected:=0;
					IF gMainAction.connected THEN
						gMainAction.homed:=0;
						gMainAction.stopped:=0;
						switch:=0;
						gFillerTyp:=AUTOMAT;
						gAxisCase:=onMOVE;
						gControl.switchToAutomat:=0;
					END_IF;
				END_IF;
			END_IF;

			//zabezpieczenia przed przejechaniem manualnym poza limit
			IF gAxisOutputs.Cart.position <= gControl.Cart.lowerLimit OR gAxisOutputs.Cart.position >= gControl.Cart.upperLimit THEN
				gControl.Cart.safeLevelStop:=1;
				IF gAxisOutputs.Cart.position >= gControl.Cart.upperLimit THEN
					gControl.Cart.onlyLeft:=1;
				ELSE
					gControl.Cart.onlyRight:=1;
				END_IF;
			ELSE
				gControl.Cart.onlyLeft:=0;
				gControl.Cart.onlyRight:=0;
				gControl.Cart.safeLevelStop:=0;
			END_IF;

			IF gAxisOutputs.Nozzle.position <= gControl.Nozzle.lowerLimit OR gAxisOutputs.Nozzle.position >= gControl.Nozzle.upperLimit THEN
				gControl.Nozzle.safeLevelStop:=1;
				IF gAxisOutputs.Nozzle.position <= gControl.Nozzle.lowerLimit THEN
					gControl.Nozzle.onlyRight:=1;
				ELSE
					gControl.Nozzle.onlyLeft:=1;
				END_IF;
			ELSE
				gControl.Nozzle.safeLevelStop:=0;
				gControl.Nozzle.onlyLeft:=0;
				gControl.Nozzle.onlyRight:=0;
			END_IF;

		AUTOMAT:
			//w przypadku naciśnięcia przycisku Stop Machine maszyna zatrzyma się po napełnieniu butelek, w state 4
			IF gControl.stop THEN
				IF gCamSeqParam.nozzle.currentStateIndex = 4 THEN
					gControl.moveVelocity:=0;
				END_IF;
			ELSE
				gControl.moveVelocity:=gControl.start AND NOT gControl.stop AND gControl.power;
			END_IF;

			//przełączenie z automatu na manual
			IF gControl.manual THEN
				gControl.moveVelocity:=0;
				gAxisCase:=DISCONNECT;
				tempVelocity:=gAxisOutputs.velocity;
				IF gMainAction.disconnected THEN
					gFillerTyp:=MANUAL;
				END_IF;
			END_IF;
	END_CASE;

END_PROGRAM

PROGRAM _EXIT
	(* Insert code here *)

END_PROGRAM
```

### Program Logical/BottleFiller/workTasks/BF_Axis (IEC)

#### Types.typ
```iecst
TYPE
	InfosTyp : 	STRUCT
		Conveyor : gControlInfoTyp;
		Cart : gControlInfoTyp;
		Nozzle : gControlInfoTyp;
	END_STRUCT;
	manualControlTyp : 	STRUCT
		errorReset : BOOL;
		start : BOOL;
		home : BOOL;
		jogNegative : BOOL;
		jogPositive : BOOL;
		stop : BOOL;
	END_STRUCT;
	axisesManagementType : 	STRUCT
		diStart : BOOL;
		diError : BOOL;
		diManual : BOOL;
		diPowerSwitch : BOOL;
		diStop : BOOL;
	END_STRUCT;
END_TYPE
```

#### Variables.var
```iecst
(*Axises*)
VAR
	MpAxisConv : MpAxisBasic;
	MpAxisCart : MpAxisBasic;
	MpAxisNozzle : MpAxisBasic;
END_VAR
(*Axis Parameters*)
VAR
	MpAxisCartParType : MpAxisBasicParType;
	MpAxisNozzleParType : MpAxisBasicParType;
	MpAxisConvParType : MpAxisBasicParType;
END_VAR
(*Cam Variables*)
VAR
	camSeq : MpAxisCamSequencer;
	camSeqNozzle : MpAxisCamSequencer;
	camNozzleParameters : MpAxisCamSequencerParType;
	configCamNozzle : McAcpAxCamAutParType;
	camParameters : MpAxisCamSequencerParType;
END_VAR
(*Other Variables*)
VAR
	timer : TON;
	stopHelper : USINT := 0;
	needUpdate : BOOL := FALSE;
	mouseEvent : BOOL := FALSE;
	homed : BOOL := FALSE; (*defines if all the axises are homed*)
END_VAR
(*global used variables*)
VAR
	axisMgmt : axisesManagementType;
	controlInfo : gAxisOutputsTyp;
	connectHelper : INT := 0;
	handleStopCart : BOOL := FALSE;
	handleStopNozzle : BOOL := FALSE;
END_VAR
```

#### Main.st
```iecst
PROGRAM _INIT
	(* Insert code here *)

	//Conveyor parameters
	MpAxisConvParType.AutoTune.Mode:=mcAXIS_TUNE_AUTOMATIC;
	MpAxisConvParType.AutoTune.MaxCurrentPercent:=80;
	MpAxisConvParType.AutoTune.MaxDistance:=30;
	MpAxisConvParType.AutoTune.SaveControllerSettings:=1;
	MpAxisConvParType.AutoTune.MaxPositionError:=30;
	//Nozzle parameters
	MpAxisNozzleParType := MpAxisConvParType;
	MpAxisNozzleParType.Homing.Position:=195;
	//Cart parameters
	MpAxisCartParType := MpAxisConvParType;

	//dynamiczna zmiana camów
	camNozzleParameters.CamSequence.Get.GetOnEnable:=1;
	camNozzleParameters.CamSequence.Get.Command:=mcGET_PAR_ACTUAL;
	camNozzleParameters.CamSequence.Data.DataAddress:=ADR(configCamNozzle);
	camNozzleParameters.CamSequence.Data.DataSize:=SIZEOF(configCamNozzle);
	camNozzleParameters.CamSequence.Set.Command:=mcSET_UPDATE_FROM_ADR;
	camNozzleParameters.CamSequence.Set.Mode:=mcAXIS_CAM_SEQ_SET_ON_UPDATE;
	MpAxisConv.AutoTune:=1;
	MpAxisCart.AutoTune:=1;
	MpAxisNozzle.AutoTune:=1;
END_PROGRAM

PROGRAM _CYCLIC
	(* Insert code here *)

	IF gControl.emergencySTOP THEN
		gAxisCase:=STANDSTILL;
		gMain:=STOP;
		gFillerTyp:=WAITING;
	END_IF;

	IF MpAxisConv.Info.AutoTuneDone THEN
		MpAxisConv.AutoTune:=0;
		MpAxisCart.AutoTune:=0;
		MpAxisNozzle.AutoTune:=0;
	END_IF;

	//deklaracja osi
	MpAxisConv(MpLink := ADR(axisConv), Enable := 1, Parameters := ADR(MpAxisConvParType));
	MpAxisCart(MpLink := ADR(axisCart), Enable := 1, Parameters := ADR(MpAxisCartParType));
	MpAxisNozzle(MpLink := ADR(axisNozzle), Enable := 1, Parameters := ADR(MpAxisNozzleParType));

	//sequence parameters
	configCamNozzle.State[3].CamID:=STRING_TO_USINT(gControl.currentBottleType);

	//Sequence declaration
	camSeq(MpLink := ADR(axisCart), Enable := 1, Parameters := ADR(camParameters), MpLinkMaster := ADR(axisConv));
	camSeqNozzle(MpLink := ADR(axisNozzle), Enable := 1, Parameters := ADR(camNozzleParameters), MpLinkMaster := ADR(axisConv));

	//conveyor management
	MpAxisConvParType.Velocity:=gAxisUpdate.Conveyor.Velocity;
	MpAxisConv.ErrorReset:=gControl.Conveyor.errorReset;
	MpAxisConv.Power:=gControl.power;
	MpAxisConv.Home:=gControl.Conveyor.home;
	MpAxisConv.Stop:=gControl.Conveyor.stop;
	MpAxisConv.JogNegative:=gControl.Conveyor.jogNegative;
	MpAxisConv.JogPositive:=gControl.Conveyor.jogPositive;

	//Cart management
	MpAxisCart.ErrorReset:=gControl.Cart.errorReset;
	MpAxisCart.Power:=gControl.power;
	MpAxisCart.Home:=gControl.Cart.home;
	MpAxisCart.Stop:=gControl.Cart.stop;
	MpAxisCart.MoveVelocity:=gControl.Cart.moveVelocity;
	MpAxisCart.JogNegative:=gControl.Cart.jogNegative;
	MpAxisCart.JogPositive:=gControl.Cart.jogPositive;

	//nozzle Management
	MpAxisNozzle.ErrorReset:=gControl.Nozzle.errorReset;
	MpAxisNozzle.Power:=gControl.power;
	MpAxisNozzle.Home:=gControl.Nozzle.home;
	MpAxisNozzle.Stop:=gControl.Nozzle.stop;
	MpAxisNozzle.JogNegative:=gControl.Nozzle.jogNegative;
	MpAxisNozzle.MoveVelocity:=gControl.Nozzle.moveVelocity;
	MpAxisNozzle.JogPositive:=gControl.Nozzle.jogPositive;

	//cam params
	camSeqNozzle.Signal1:=gCamSeqParam.nozzle.signal1;

	//aktualizacja predkosci po kliknieciu przycisku manipulujacego predkoscia o +-5%
	IF gControl.partVelUpd THEN
		MpAxisConvParType.Velocity:=gAxisUpdate.Conveyor.Velocity;
		MpAxisConv.Update:=1;
		gControl.partVelUpd:=0;
	END_IF;

	//aktualizacja osi po zmianie parametrów
	IF gControl.needUpdate THEN
		//conveyor
		IF gControl.manual THEN
			MpAxisConvParType.Velocity:=gAxisUpdate.Conveyor.Velocity;
		ELSE
			MpAxisConvParType.Velocity:=STRING_TO_UINT(gAxisUpdate.staticVelocity);
			gAxisUpdate.Conveyor.Velocity:=STRING_TO_UINT(gAxisUpdate.staticVelocity);
		END_IF;

		MpAxisConvParType.Jog.LimitPosition.FirstPosition:=gAxisUpdate.Conveyor.FirstPosition;
		MpAxisConvParType.Jog.LimitPosition.LastPosition:=gAxisUpdate.Conveyor.LastPosition;
		MpAxisConvParType.Position:=gAxisUpdate.Conveyor.Position;
		MpAxisConvParType.Jog.Velocity:=gAxisUpdate.Conveyor.Velocity;

		//velocity range update
		gControl.maxVelocity:= 1.2 * STRING_TO_UINT(gAxisUpdate.staticVelocity);
		gControl.minVelocity:= 0.8 * STRING_TO_UINT(gAxisUpdate.staticVelocity);
		gControl.part:=0.05 * STRING_TO_UINT(gAxisUpdate.staticVelocity);
		gControl.incVisible:=1;
		gControl.decVisible:=1;

		//cart
		MpAxisCartParType.Jog.LimitPosition.FirstPosition:=gAxisUpdate.Cart.FirstPosition;
		MpAxisCartParType.Jog.LimitPosition.LastPosition:=gAxisUpdate.Cart.LastPosition;
		MpAxisCartParType.Position:=gAxisUpdate.Cart.Position;
		MpAxisCartParType.Jog.Velocity:=gAxisUpdate.Conveyor.Velocity;
		MpAxisCartParType.Velocity:=gAxisUpdate.Conveyor.Velocity;

		//nozzle
		MpAxisNozzleParType.Jog.LimitPosition.FirstPosition:=gAxisUpdate.Nozzle.FirstPosition;
		MpAxisNozzleParType.Jog.LimitPosition.LastPosition:=gAxisUpdate.Nozzle.LastPosition;
		MpAxisNozzleParType.Position:=gAxisUpdate.Nozzle.Position;
		MpAxisNozzleParType.Jog.Velocity:=gAxisUpdate.Conveyor.Velocity;
		MpAxisNozzleParType.Velocity:=gAxisUpdate.Conveyor.Velocity;

		camParameters.Offset.Velocity:=gAxisUpdate.Conveyor.Velocity+30;
		camNozzleParameters.Offset.Velocity:=gAxisUpdate.Conveyor.Velocity+30;

		MpAxisNozzle.Update:=1;
		MpAxisConv.Update:=1;
		MpAxisCart.Update:=1;
		gControl.needUpdate:=0;
	END_IF;

	CASE gAxisCase OF
		HOLDON:
			MpAxisCart.Stop:=1;
			MpAxisConv.Stop:=1;
			MpAxisNozzle.Stop:=1;
			IF MpAxisConv.Stopped AND MpAxisNozzle.Stopped AND MpAxisCart.Stopped THEN
				MpAxisCart.Stop:=0;
				MpAxisConv.Stop:=0;
				MpAxisNozzle.Stop:=0;
				stopHelper:=1;
			END_IF;
			IF stopHelper=1 THEN
				IF  MpAxisConv.Info.PLCopenState = mcAXIS_STANDSTILL AND MpAxisCart.Info.PLCopenState = mcAXIS_STANDSTILL AND MpAxisNozzle.Info.PLCopenState = mcAXIS_STANDSTILL THEN
					gMainAction.stopped:=1;
					stopHelper:=0;
				END_IF;
			END_IF;

		POWERED:
			IF (gControl.power AND NOT gAxisOutputs.Conveyor.error) THEN
				//power on axis
				MpAxisCart.Power:=1;
				MpAxisConv.Power:=1;
				MpAxisNozzle.Power:=1;

				IF MpAxisCart.PowerOn AND MpAxisConv.PowerOn AND MpAxisNozzle.PowerOn THEN
					gMainAction.powered:=1;
				END_IF;

			END_IF;

		HOMING:
			gControl.bottleCnt:=0;
			IF MpAxisCart.Info.PLCopenState = mcAXIS_STANDSTILL THEN
				MpAxisConv.Home:=1;
				MpAxisNozzle.Home:=1;
				MpAxisCart.Home:=1;

			END_IF;

			IF MpAxisCart.Info.PLCopenState = mcAXIS_HOMING THEN
				connectHelper:=15;
			END_IF;

			IF connectHelper=15 AND MpAxisCart.Info.PLCopenState = mcAXIS_STANDSTILL THEN
				gMainAction.homed:=1;
			END_IF;

		STANDSTILL:
			IF gControl.start THEN
				IF gControl.manual THEN
					gAxisCase:=onMOVE;
				ELSE
					IF gControl.inCam THEN
						gAxisCase:=onMOVE;
					ELSE
						gAxisCase:=CONNECT;
					END_IF;

				END_IF;
			END_IF;

		CONNECT:
			camSeq.EndSequence:=0;
			camSeqNozzle.EndSequence:=0;

			IF NOT gControl.manual AND NOT gControl.switchToAutomat THEN
				camSeq.StartSequence:=1;
				camSeqNozzle.StartSequence:=1;
			ELSE
				IF camSeq.Error THEN
					camSeq.ErrorReset:=1;
					timer.IN:=TRUE;
					timer.PT:=t#100ms;
					IF timer.Q THEN
						timer.IN:=FALSE;
						camSeq.StartSequence:=0;
					END_IF;
				END_IF;
				IF camSeq.StartSequence=0 THEN

					timer.IN:=TRUE;
					timer.PT:=t#200ms;
					IF timer.Q THEN
						timer.IN:=FALSE;
						camSeq.StartSequence:=1;
						camSeqNozzle.StartSequence:=1;
					END_IF;
				END_IF;

			END_IF;
			IF camSeq.InCam AND camSeqNozzle.InCam  THEN
				camSeq.Signal1:=1;
				gMainAction.connected:=1;
				connectHelper:=0;
			END_IF;

		DISCONNECT:
			gMainAction.connected:=0;
			MpAxisConv.MoveVelocity:=0;
			camSeq.Signal1:=0;
			camSeqNozzle.Signal1:=0;
			camSeq.StartSequence:=0;
			camSeq.EndSequence:=1;
			camSeqNozzle.StartSequence:=0;
			camSeqNozzle.EndSequence:=1;
			IF NOT (camSeq.Running AND camSeqNozzle.Running) THEN
				gMainAction.disconnected:=1;
			END_IF;

		onMOVE:
			//karetka
			IF mouseEvent THEN
				IF gControl.Cart.safeLevelStop THEN
					gControl.Cart.stop:=gControl.Cart.safeLevelStop;
					IF MpAxisCartParType.Direction = 1 AND MpAxisCart.Position >= gControl.Cart.upperLimit THEN
						gControl.Cart.safeLevelStop:=0;
						gControl.Cart.stop:=0;
					ELSIF MpAxisCartParType.Direction = 0 AND MpAxisCart.Position <= gControl.Cart.lowerLimit THEN
						gControl.Cart.safeLevelStop:=0;
						gControl.Cart.stop:=0;
					END_IF;
				END_IF;

				IF gControl.Nozzle.safeLevelStop THEN
					gControl.Nozzle.stop:=gControl.Nozzle.safeLevelStop;
					IF MpAxisNozzleParType.Direction = 1 AND MpAxisNozzle.Position >= gControl.Nozzle.upperLimit THEN
						gControl.Nozzle.safeLevelStop:=0;
						gControl.Nozzle.stop:=0;
					ELSIF MpAxisNozzleParType.Direction = 0 AND MpAxisNozzle.Position <= gControl.Nozzle.lowerLimit THEN
						gControl.Nozzle.safeLevelStop:=0;
						gControl.Nozzle.stop:=0;
					END_IF;
				END_IF;

				MpAxisConv.MoveVelocity:=gControl.moveVelocity;

				IF gControl.Cart.onlyRight AND MpAxisCartParType.Direction = 0 THEN
					gControl.Cart.stop:=0;
					MpAxisCart.MoveVelocity:=gControl.Cart.moveVelocity;
				END_IF;

				IF gControl.Cart.onlyLeft AND MpAxisCartParType.Direction = 1 THEN
					gControl.Cart.stop:=0;
					MpAxisCart.MoveVelocity:=gControl.Cart.moveVelocity;
				END_IF;

				IF NOT gControl.Cart.onlyLeft AND NOT gControl.Cart.onlyRight THEN
					MpAxisCart.MoveVelocity:= NOT gControl.Cart.safeLevelStop AND gControl.Cart.moveVelocity;
				END_IF;

				//nozzle
				IF gControl.Nozzle.onlyRight AND MpAxisNozzleParType.Direction = 0 THEN
					gControl.Nozzle.stop:=0;
					MpAxisNozzle.MoveVelocity:=gControl.Nozzle.moveVelocity;
				END_IF;

				IF gControl.Nozzle.onlyLeft AND MpAxisNozzleParType.Direction = 1 THEN
					gControl.Nozzle.stop:=0;
					MpAxisNozzle.MoveVelocity:=gControl.Nozzle.moveVelocity;
				END_IF;

				IF NOT gControl.Nozzle.onlyLeft AND NOT gControl.Nozzle.onlyRight THEN
					MpAxisNozzle.MoveVelocity:= NOT gControl.Nozzle.safeLevelStop AND gControl.Nozzle.moveVelocity;
				END_IF;
			ELSE
				MpAxisConv.MoveVelocity:=gControl.moveVelocity;
				MpAxisConv.JogNegative:=gControl.Conveyor.jogNegative;
				MpAxisConv.JogPositive:=gControl.Conveyor.jogPositive;
				MpAxisCart.JogNegative:=gControl.Cart.jogNegative;
				MpAxisCart.JogPositive:=gControl.Cart.jogPositive;
				MpAxisNozzle.JogNegative:=gControl.Nozzle.jogNegative;
				MpAxisNozzle.JogPositive:=gControl.Nozzle.jogPositive;
			END_IF;
			IF MpAxisConv.Position > 0 THEN
				gMainAction.homed:=0;
			END_IF;

	END_CASE;

	controlInfo.Conveyor.error:=MpAxisConv.Error;
	controlInfo.Conveyor.isHomed:=MpAxisConv.IsHomed;
	controlInfo.Conveyor.isPowered:=MpAxisConv.PowerOn;
	controlInfo.Conveyor.position:=LREAL_TO_REAL(MpAxisConv.Position);
	controlInfo.Conveyor.velocity:=MpAxisConv.Velocity;
	controlInfo.Conveyor.updateDone:=MpAxisConv.UpdateDone;
	controlInfo.Conveyor.MoveActive:=MpAxisConv.Info.Jogging;

	controlInfo.Cart.error:=MpAxisCart.Error;
	controlInfo.Cart.isHomed:=MpAxisCart.IsHomed;
	controlInfo.Cart.isPowered:=MpAxisCart.PowerOn;
	controlInfo.Cart.position:=LREAL_TO_REAL(MpAxisCart.Position);
	controlInfo.Cart.velocity:=MpAxisCart.Velocity;
	controlInfo.Cart.updateDone:=MpAxisCart.UpdateDone;
	controlInfo.Cart.MoveActive:=MpAxisCart.Info.Jogging;

	controlInfo.Nozzle.error:=MpAxisNozzle.Error;
	controlInfo.Nozzle.isHomed:=MpAxisNozzle.IsHomed;
	controlInfo.Nozzle.isPowered:=MpAxisNozzle.PowerOn;
	controlInfo.Nozzle.position:=LREAL_TO_REAL(MpAxisNozzle.Position);
	controlInfo.Nozzle.velocity:=MpAxisNozzle.Velocity;
	controlInfo.Nozzle.updateDone:=MpAxisNozzle.UpdateDone;
	controlInfo.Nozzle.MoveActive:=MpAxisNozzle.Info.Jogging;

	controlInfo.velocity:=MpAxisConvParType.Velocity;

	gCamSeqParam.cart.currentStateIndex:=camSeq.ActualStateIndex;
	gCamSeqParam.nozzle.currentStateIndex:=camSeqNozzle.ActualStateIndex;

	gAxisOutputs:=controlInfo;

	IF camSeq.OffsetDone THEN
		camSeq.OffsetShift:=0;
	END_IF;
	IF camSeqNozzle.OffsetDone THEN
		camSeqNozzle.OffsetShift:=0;
	END_IF;

	IF camSeqNozzle.UpdateDone THEN
		camSeqNozzle.Update:=0;
	END_IF;
	IF MpAxisConv.UpdateDone THEN
		MpAxisConv.Update:=0;
	END_IF;
	IF MpAxisNozzle.UpdateDone THEN
		MpAxisNozzle.Update:=0;
	END_IF;
	IF MpAxisCart.UpdateDone THEN
		MpAxisCart.Update:=0;
	END_IF;
	timer();
END_PROGRAM

PROGRAM _EXIT
	(* Insert code here *)

END_PROGRAM
```

### Program Logical/BottleFiller/workTasks/Program (ANSIC)

#### Variables.var
```iecst
VAR
	BF_MpAlarm : MpAlarmXCore;
	caseError : errorCaseEnum;
	resetError : USINT := 0;
	error : INT := 0;
END_VAR
```

#### Main.c
```c
#include <bur/plctypes.h>

#ifdef _DEFAULT_INCLUDES
	#include <AsDefault.h>
	#include <brsystem.h>
#endif
void _INIT ProgramInit(void)
{

}

void _CYCLIC ProgramCyclic(void)
{
	BF_MpAlarm.MpLink=&(gAlarmXCore);
	BF_MpAlarm.Enable=1;

	gControl.moveVelocity =(gControl.moveVelocity==1 && error==0);
	gControl.Conveyor.jogNegative =(gControl.Conveyor.jogNegative==1 && error==0);
	gControl.Conveyor.jogPositive =(gControl.Conveyor.jogPositive==1 & error==0);
	gControl.Cart.jogNegative =(gControl.Cart.jogNegative==1 && error==0);
	gControl.Cart.jogPositive =(gControl.Cart.jogPositive==1 && error==0);
	gControl.Cart.moveVelocity =(gControl.Cart.moveVelocity==1 && error==0);
	gControl.Nozzle.jogNegative =(gControl.Nozzle.jogNegative==1 && error==0);
	gControl.Nozzle.jogPositive =(gControl.Nozzle.jogPositive==1 && error==0);
	gControl.Nozzle.moveVelocity =(gControl.Nozzle.moveVelocity==1 && error==0);

	switch (caseError)
	{
	case noError:
	if (gControl.start &&  !(gControl.power))
	{
		MpAlarmXSet(&gAlarmXCore, 'noPower');
		caseError=inError;
		error=1;
	}

	if (BF_MpAlarm.PendingAlarms != 0)
	{
	caseError=inError;
	error=1;
	}
	break;

	case inError:
	gAxisCase=WAIT;
	gMain=ERROR;
	gFillerTyp=WAITING;
	if( !(gControl.start && !(gControl.power)))
	MpAlarmXReset(&(gAlarmXCore), 'noPower');

	if (resetError != 0 )
	caseError=handleError;

	if (BF_MpAlarm.PendingAlarms==0)
	{
	caseError=noError;
	error=0;
	gMain=WORK;
	gFillerTyp=MANUAL;
	gAxisCase=onMOVE;
	}
	break;

	case handleError:
	if (resetError==1)
	{
	gControl.Nozzle.errorReset=1;
	if (!(gAxisOutputs.Nozzle.error))
	{
	gControl.Nozzle.errorReset=0;
	caseError=inError;
	resetError=0;
	}
	}
	if (resetError==2)
	{
	gControl.Conveyor.errorReset=1;
	if (!(gAxisOutputs.Conveyor.error))
	{
	gControl.Conveyor.errorReset=0;
	caseError=inError;
	resetError=0;
	}
	}
	if (resetError==3)
	{
	gControl.Cart.errorReset=1;
	if (!(gAxisOutputs.Cart.error))
	{
	gControl.Cart.errorReset=0;
	caseError=inError;
	resetError=0;
	}
	}
	break;
	}

}

void _EXIT ProgramExit(void)
{

}
```

### Program Logical/BottleFiller/workTasks/BF_Alarm (IEC)

#### Types.typ
```iecst
TYPE
	errorCaseEnum :
		(
		noError,
		handleError,
		inError
		);
END_TYPE
```

#### Variables.var
```iecst
VAR
	BF_MpAlarm : MpAlarmXCore;
	resetError : USINT := 0;
	error : BOOL := FALSE;
END_VAR
```

#### Main.st
```iecst
PROGRAM _INIT
	(* Insert code here *)

END_PROGRAM

PROGRAM _CYCLIC
	(* Insert code here *)
	BF_MpAlarm(MpLink:=ADR(gBFAlarmXCore), Enable:=TRUE);

	gControl.moveVelocity:= gControl.moveVelocity AND NOT error;
	gControl.Conveyor.jogNegative:= gControl.Conveyor.jogNegative AND NOT error;
	gControl.Conveyor.jogPositive:= gControl.Conveyor.jogPositive AND NOT error;
	gControl.Cart.jogNegative := gControl.Cart.jogNegative AND NOT error;
	gControl.Cart.jogPositive := gControl.Cart.jogPositive AND NOT error;
	gControl.Cart.moveVelocity := gControl.Cart.moveVelocity AND NOT error;
	gControl.Nozzle.jogNegative := gControl.Nozzle.jogNegative AND NOT error;
	gControl.Nozzle.jogPositive := gControl.Nozzle.jogPositive AND NOT error;
	gControl.Nozzle.moveVelocity := gControl.Nozzle.moveVelocity AND NOT error;

	CASE gCaseError OF
		noError:
			IF gControl.start AND NOT gControl.power THEN
				MpAlarmXSet(gBFAlarmXCore, 'noPower');
				gCaseError:=inError;
				error:=1;
			END_IF;
			IF gControl.emergencySTOP THEN
				MpAlarmXSet(gBFAlarmXCore, 'emergency');
				gCaseError:=inError;
				error:=1;
			END_IF;
			IF BF_MpAlarm.PendingAlarms <> 0 THEN
				gCaseError:=inError;

				error:=1;
			END_IF;

		inError:
			gAxisCase:=WAIT;
			gMain:=ERROR;
			gFillerTyp:=WAITING;
			IF NOT(gControl.start AND NOT gControl.power) THEN
				MpAlarmXReset(gBFAlarmXCore, 'noPower');
			END_IF;
			IF NOT(gControl.emergencySTOP) THEN
				MpAlarmXReset(gBFAlarmXCore, 'emergency');
			END_IF;

			IF resetError <> 0 THEN
				gCaseError:=handleError;
			END_IF;

			IF BF_MpAlarm.PendingAlarms=0 THEN

				error:=0;
				gMain:=WORK;
				IF temp THEN
					gAxisCase:=DISCONNECT;
					IF gMainAction.disconnected THEN
						gAxisCase:=CONNECT;
					END_IF;
					IF gMainAction.connected THEN
						gAxisCase:=onMOVE;
						gFillerTyp:=AUTOMAT;
						gCaseError:=noError;
					END_IF;
				ELSE
					gFillerTyp:=MANUAL;
					gAxisCase:=onMOVE;
					gCaseError:=noError;
				END_IF;

			END_IF;

		handleError:
			IF resetError = 1 THEN
				gControl.Nozzle.errorReset:=1;
				IF NOT gAxisOutputs.Nozzle.error THEN
					gControl.Nozzle.errorReset:=0;
					gCaseError:=inError;
					resetError:=0;
				END_IF;
			END_IF;
			IF resetError = 2 THEN
				gControl.Conveyor.errorReset:=1;
				IF NOT gAxisOutputs.Conveyor.error THEN
					gControl.Conveyor.errorReset:=0;
					gCaseError:=inError;
					resetError:=0;
				END_IF;
			END_IF;
			IF resetError = 3 THEN
				gControl.Cart.errorReset:=1;
				IF NOT gAxisOutputs.Cart.error THEN
					gControl.Cart.errorReset:=0;
					gCaseError:=inError;
					resetError:=0;
				END_IF;
			END_IF;

	END_CASE;

END_PROGRAM

PROGRAM _EXIT
	(* Insert code here *)
	 BF_MpAlarm(Enable:=0);
END_PROGRAM
```

### Types.typ - not listed in the package file held
```iecst
TYPE
	bottleFillerRecipeEnum : 	STRUCT
		diPumpSpeedFlow : INT := 0;
		diVelocity : INT := 0;
		diSpeedProfile : INT := 0;
		diBottleShape : INT := 0;
	END_STRUCT;
	FillerEnum :
		( (*Every possible case*)
		DISABLED,
		STOP,
		SERVICE,
		INIT,
		AUTOMAT,
		ERROR
		);
END_TYPE
```

### Variables.var - not listed in the package file held
```iecst
(*case machine*)
VAR
	FillerTyp : FillerEnum;
	bottleFillerRecipeTyp : bottleFillerRecipeEnum;
END_VAR
(*digital inputs*)
VAR
	diError : BOOL;
	diManual : BOOL := FALSE; (*Determine if machine works automatically or needs manual control*)
	diStop : BOOL := FALSE; (*Stop switch*)
	diStart : BOOL := FALSE; (*Start switch*)
	diPowerSwitch : BOOL := FALSE; (*Power on switch*)
	diLiquidLevel : REAL := 100;
	diConveyorHomingSwitch : BOOL := FALSE; (*Sensor detecting conveyor at homing position*)
	diNozzleHomingSwitch : BOOL := FALSE; (*Sensor detecting nozzle at homing position*)
	diCartHomingSwitch : BOOL := FALSE; (*Sensor detecting cart at homing position*)
	diBottleDetection : BOOL := FALSE; (*Sensor detecting presence of a bottle*)
END_VAR
(*digital outputs*)
VAR
	doPumpRelay : INT; (*Output controlling the pump building pressure for liquid flow*)
	doValveRelay : BOOL; (*Output controlling the liquid valve opening*)
END_VAR
(*analog outputs*)
VAR
	aoPumpFlowSpeed : ARRAY[0..100] OF INT; (*Datapoint in percentage to the pump system about liquid flow speed in percent*)
END_VAR
(*other variables*)
VAR
	roleInfo : MpUserXMgrUIRoleInfoType;
	MpBFRecipeXml : MpRecipeXml;
	MpBFRecipeRegPar : MpRecipeRegPar; (*MpBFRecipeHMI : MpRecipeUI;
	UISetup : MpRecipeUISetupType;
	MpRecipeUIConnectType : MpRecipeUIConnectType;*)
	MpAxisConvParType : MpAxisBasicParType;
	MpAxisConv : MpAxisBasic;
	MpAxisCart : MpAxisBasic;
	MpAxisNozzle : MpAxisBasic;
END_VAR
```

### Main.st - not listed in the package file held
```iecst
PROGRAM _INIT
	(* Insert code here *)
	 FillerTyp:=DISABLED;
END_PROGRAM

PROGRAM _CYCLIC
	(* Insert code here *)
	MpBFRecipeXml(MpLink := ADR(BFRecipe) , Enable := 1, DeviceName := ADR('USER') , FileName := ADR('BottleFillerRecipe'));
	MpBFRecipeRegPar(MpLink := ADR(BFRecipe), Enable := 1, PVName := ADR('BootleFiller:bottleFillerRecipeTyp'));
	//MpBFRecipeHMI(MpLink := ADR(BFRecipe), Enable := 1 , ErrorReset := , UISetup := ADR(UISetup) , UIConnect := ADR(MpRecipeUIConnectType));
	MpAxisConvParType.AutoTune.Mode:=mcAXIS_TUNE_AUTOMATIC;
	MpAxisConvParType.AutoTune.MaxCurrentPercent:=80;
	MpAxisConvParType.AutoTune.MaxDistance:=30;
	MpAxisConvParType.AutoTune.MaxPositionError:=30;
	MpAxisConv(MpLink := ADR(axisConv), Enable := 1, Parameters := ADR(MpAxisConvParType) ,   AutoTune := 1);
	MpAxisCart(MpLink := ADR(axisCart), Enable := 1, Parameters := ADR(MpAxisConvParType) ,   AutoTune := 1);
	MpAxisNozzle(MpLink := ADR(axisNozzle), Enable := 1, Parameters := ADR(MpAxisConvParType) ,  AutoTune := 1);

	MpBFRecipeXml();
	//MpBFRecipeHMI();
	CASE FillerTyp OF
		DISABLED:
			diStart:=0;
			diStop:=0;

			IF diPowerSwitch THEN
				FillerTyp:=INIT;
			END_IF;

		INIT:
			//procedury początkowe; home, kierunek
			IF diStart AND NOT diStop AND NOT diError THEN
				IF diManual THEN
					FillerTyp:=SERVICE;
				ELSE
					FillerTyp:= AUTOMAT;
				END_IF;
			END_IF;

		AUTOMAT:

		SERVICE:

		ERROR:

		STOP:

	END_CASE;

END_PROGRAM

PROGRAM _EXIT
	(* Insert code here *)

END_PROGRAM
```

- Visualisation Logical/mappView (not shown)

### Data object Logical/b1_Nozzle (Cam)

#### b1_Nozzle.cam - Cam for mapp Motion
```
CamProfile (NcSwId=ACP10, MasterAxisVelocity=1, MasterAxisAcceleration=0, DefaultCurveType=Polynomial5, MathematicalNotation=true)
  FixPoint (x=0, IsMathX=true, y=0, IsDefinedDy=false, Dy=0, IsMathDy=true, IsDefinedDdy=false, Ddy=0, IsMathDdy=true, IsDefinedDddy=false, Dddy=0, IsMathDddy=true)
  FixPoint (x=1, IsMathX=true, y=1, IsDefinedDy=true, Dy=0, IsMathDy=true, IsDefinedDdy=true, Ddy=0, IsMathDdy=true, IsDefinedDddy=false, Dddy=0, IsMathDddy=true)
  Synchronline:
    LeftBoundary (IsFix=true, x=0.4, IsMathX=true, y=0.6)
    RightBoundary (IsFix=true, x=0.7, IsMathX=true, y=0.8)
    Gradient (Numerator=2, Denominator=3, IsMath=false, IsFix=false)
  Curve (Type=Polynomial5)
    LeftBoundary (IsDefinedDdy=false, Ddy=0, IsMathDdy=true, IsDefinedDddy=false, Dddy=0, IsMathDddy=true)
    RightBoundary (IsDefinedDdy=false, Ddy=0, IsMathDdy=true, IsDefinedDddy=false, Dddy=0, IsMathDddy=true)
    Spline3 (IsContinuous4Derivative=false, IsDefinedSaddlePoint=false, IsDefinedLineAs2ndSegment=false, IsDefinedSlopeOfLine=false, SlopeOfLine=0, IsMathSlopeOfLine=true)
    Supremum (y=1.7e+308, Dy=1.7e+308, IsMathDy=true, Ddy=1.7e+308, IsMathDdy=true, Dddy=1.7e+308, IsMathDddy=true)
    Infimum (y=-1.7e+308, Dy=-1.7e+308, IsMathDy=true, Ddy=-1.7e+308, IsMathDdy=true, Dddy=-1.7e+308, IsMathDddy=true)
  Curve (Type=Polynomial5)
    LeftBoundary (IsDefinedDdy=false, Ddy=0, IsMathDdy=true, IsDefinedDddy=false, Dddy=0, IsMathDddy=true)
    RightBoundary (IsDefinedDdy=false, Ddy=0, IsMathDdy=true, IsDefinedDddy=false, Dddy=0, IsMathDddy=true)
    Spline3 (IsContinuous4Derivative=false, IsDefinedSaddlePoint=false, IsDefinedLineAs2ndSegment=false, IsDefinedSlopeOfLine=false, SlopeOfLine=0, IsMathSlopeOfLine=true)
    Supremum (y=1.7e+308, Dy=1.7e+308, IsMathDy=true, Ddy=1.7e+308, IsMathDdy=true, Dddy=1.7e+308, IsMathDddy=true)
    Infimum (y=-1.7e+308, Dy=-1.7e+308, IsMathDy=true, Ddy=-1.7e+308, IsMathDdy=true, Dddy=-1.7e+308, IsMathDddy=true)
  Cam (LeftBoundaryIndex=0, RightBoundaryIndex=3)
    Supremum (y=1.7e+308, Dy=1.7e+308, IsMathDy=true, Ddy=1.7e+308, IsMathDdy=true, Dddy=1.7e+308, IsMathDddy=true)
    Infimum (y=-1.7e+308, Dy=-1.7e+308, IsMathDy=true, Ddy=-1.7e+308, IsMathDdy=true, Dddy=1.7e+308, IsMathDddy=true)
  ChartExtensions
```

### Data object Logical/b2_Nozzle (Cam)

#### b2_Nozzle.cam - Cam for mapp Motion
```
CamProfile (NcSwId=ACP10, MasterAxisVelocity=1, MasterAxisAcceleration=0, DefaultCurveType=Polynomial5, MathematicalNotation=true)
  FixPoint (x=0, IsMathX=true, y=0, IsDefinedDy=false, Dy=0, IsMathDy=true, IsDefinedDdy=false, Ddy=0, IsMathDdy=true, IsDefinedDddy=false, Dddy=0, IsMathDddy=true)
  FixPoint (x=1, IsMathX=true, y=1, IsDefinedDy=false, Dy=0, IsMathDy=true, IsDefinedDdy=false, Ddy=0, IsMathDdy=true, IsDefinedDddy=false, Dddy=0, IsMathDddy=true)
  Synchronline:
    LeftBoundary (IsFix=true, x=1e-06, IsMathX=true, y=1e-06)
    RightBoundary (IsFix=true, x=0.2, IsMathX=true, y=0.175)
    Gradient (Numerator=874999, Denominator=1000000, IsMath=false, IsFix=false)
  Synchronline:
    LeftBoundary (IsFix=true, x=0.25, IsMathX=true, y=0.225)
    RightBoundary (IsFix=true, x=0.45, IsMathX=true, y=0.375)
    Gradient (Numerator=3, Denominator=4, IsMath=false, IsFix=false)
  Synchronline:
    LeftBoundary (IsFix=true, x=0.5, IsMathX=true, y=0.425)
    RightBoundary (IsFix=true, x=0.7, IsMathX=true, y=0.575)
    Gradient (Numerator=3, Denominator=4, IsMath=false, IsFix=false)
  Curve (Type=Polynomial5)
    LeftBoundary (IsDefinedDdy=false, Ddy=0, IsMathDdy=true, IsDefinedDddy=false, Dddy=0, IsMathDddy=true)
    RightBoundary (IsDefinedDdy=false, Ddy=0, IsMathDdy=true, IsDefinedDddy=false, Dddy=0, IsMathDddy=true)
    Spline3 (IsContinuous4Derivative=false, IsDefinedSaddlePoint=false, IsDefinedLineAs2ndSegment=false, IsDefinedSlopeOfLine=false, SlopeOfLine=0, IsMathSlopeOfLine=true)
    Supremum (y=1.7e+308, Dy=1.7e+308, IsMathDy=true, Ddy=1.7e+308, IsMathDdy=true, Dddy=1.7e+308, IsMathDddy=true)
    Infimum (y=-1.7e+308, Dy=-1.7e+308, IsMathDy=true, Ddy=-1.7e+308, IsMathDdy=true, Dddy=-1.7e+308, IsMathDddy=true)
  Curve (Type=Polynomial5)
    LeftBoundary (IsDefinedDdy=false, Ddy=0, IsMathDdy=true, IsDefinedDddy=false, Dddy=0, IsMathDddy=true)
    RightBoundary (IsDefinedDdy=false, Ddy=0, IsMathDdy=true, IsDefinedDddy=false, Dddy=0, IsMathDddy=true)
    Spline3 (IsContinuous4Derivative=false, IsDefinedSaddlePoint=false, IsDefinedLineAs2ndSegment=false, IsDefinedSlopeOfLine=false, SlopeOfLine=0, IsMathSlopeOfLine=true)
    Supremum (y=1.7e+308, Dy=1.7e+308, IsMathDy=true, Ddy=1.7e+308, IsMathDdy=true, Dddy=1.7e+308, IsMathDddy=true)
    Infimum (y=-1.7e+308, Dy=-1.7e+308, IsMathDy=true, Ddy=-1.7e+308, IsMathDdy=true, Dddy=-1.7e+308, IsMathDddy=true)
  Curve (Type=Polynomial5)
    LeftBoundary (IsDefinedDdy=false, Ddy=0, IsMathDdy=true, IsDefinedDddy=false, Dddy=0, IsMathDddy=true)
    RightBoundary (IsDefinedDdy=false, Ddy=0, IsMathDdy=true, IsDefinedDddy=false, Dddy=0, IsMathDddy=true)
    Spline3 (IsContinuous4Derivative=false, IsDefinedSaddlePoint=false, IsDefinedLineAs2ndSegment=false, IsDefinedSlopeOfLine=false, SlopeOfLine=0, IsMathSlopeOfLine=true)
    Supremum (y=1.7e+308, Dy=1.7e+308, IsMathDy=true, Ddy=1.7e+308, IsMathDdy=true, Dddy=1.7e+308, IsMathDddy=true)
    Infimum (y=-1.7e+308, Dy=-1.7e+308, IsMathDy=true, Ddy=-1.7e+308, IsMathDdy=true, Dddy=-1.7e+308, IsMathDddy=true)
  Curve (Type=Polynomial5)
    LeftBoundary (IsDefinedDdy=false, Ddy=0, IsMathDdy=true, IsDefinedDddy=false, Dddy=0, IsMathDddy=true)
    RightBoundary (IsDefinedDdy=false, Ddy=0, IsMathDdy=true, IsDefinedDddy=false, Dddy=0, IsMathDddy=true)
    Spline3 (IsContinuous4Derivative=false, IsDefinedSaddlePoint=false, IsDefinedLineAs2ndSegment=false, IsDefinedSlopeOfLine=false, SlopeOfLine=0, IsMathSlopeOfLine=true)
    Supremum (y=1.7e+308, Dy=1.7e+308, IsMathDy=true, Ddy=1.7e+308, IsMathDdy=true, Dddy=1.7e+308, IsMathDddy=true)
    Infimum (y=-1.7e+308, Dy=-1.7e+308, IsMathDy=true, Ddy=-1.7e+308, IsMathDdy=true, Dddy=-1.7e+308, IsMathDddy=true)
  Cam (LeftBoundaryIndex=0, RightBoundaryIndex=7)
    Supremum (y=1.7e+308, Dy=1.7e+308, IsMathDy=true, Ddy=1.7e+308, IsMathDdy=true, Dddy=1.7e+308, IsMathDddy=true)
    Infimum (y=-1.7e+308, Dy=-1.7e+308, IsMathDy=true, Ddy=-1.7e+308, IsMathDdy=true, Dddy=1.7e+308, IsMathDddy=true)
  ChartExtensions
```

### Data object Logical/b3_Nozzle (Cam)

#### b3_Nozzle.cam - Cam for mapp Motion
```
CamProfile (NcSwId=ACP10, MasterAxisVelocity=1, MasterAxisAcceleration=0, DefaultCurveType=Polynomial5, MathematicalNotation=true)
  FixPoint (x=0, IsMathX=true, y=0, IsDefinedDy=false, Dy=0, IsMathDy=true, IsDefinedDdy=false, Ddy=0, IsMathDdy=true, IsDefinedDddy=false, Dddy=0, IsMathDddy=true)
  FixPoint (x=1, IsMathX=true, y=1, IsDefinedDy=false, Dy=0, IsMathDy=true, IsDefinedDdy=false, Ddy=0, IsMathDdy=true, IsDefinedDddy=false, Dddy=0, IsMathDddy=true)
  Synchronline:
    LeftBoundary (IsFix=true, x=1e-06, IsMathX=true, y=1e-06)
    RightBoundary (IsFix=true, x=0.5, IsMathX=true, y=0.4)
    Gradient (Numerator=4, Denominator=5, IsMath=false, IsFix=false)
  Synchronline:
    LeftBoundary (IsFix=true, x=0.685, IsMathX=true, y=0.725)
    RightBoundary (IsFix=true, x=0.875, IsMathX=true, y=0.9)
    Gradient (Numerator=35, Denominator=38, IsMath=false, IsFix=false)
  Curve (Type=Polynomial5)
    LeftBoundary (IsDefinedDdy=false, Ddy=0, IsMathDdy=true, IsDefinedDddy=false, Dddy=0, IsMathDddy=true)
    RightBoundary (IsDefinedDdy=false, Ddy=0, IsMathDdy=true, IsDefinedDddy=false, Dddy=0, IsMathDddy=true)
    Spline3 (IsContinuous4Derivative=false, IsDefinedSaddlePoint=false, IsDefinedLineAs2ndSegment=false, IsDefinedSlopeOfLine=false, SlopeOfLine=0, IsMathSlopeOfLine=true)
    Supremum (y=1.7e+308, Dy=1.7e+308, IsMathDy=true, Ddy=1.7e+308, IsMathDdy=true, Dddy=1.7e+308, IsMathDddy=true)
    Infimum (y=-1.7e+308, Dy=-1.7e+308, IsMathDy=true, Ddy=-1.7e+308, IsMathDdy=true, Dddy=-1.7e+308, IsMathDddy=true)
  Curve (Type=Polynomial5)
    LeftBoundary (IsDefinedDdy=false, Ddy=0, IsMathDdy=true, IsDefinedDddy=false, Dddy=0, IsMathDddy=true)
    RightBoundary (IsDefinedDdy=false, Ddy=0, IsMathDdy=true, IsDefinedDddy=false, Dddy=0, IsMathDddy=true)
    Spline3 (IsContinuous4Derivative=false, IsDefinedSaddlePoint=false, IsDefinedLineAs2ndSegment=false, IsDefinedSlopeOfLine=false, SlopeOfLine=0, IsMathSlopeOfLine=true)
    Supremum (y=1.7e+308, Dy=1.7e+308, IsMathDy=true, Ddy=1.7e+308, IsMathDdy=true, Dddy=1.7e+308, IsMathDddy=true)
    Infimum (y=-1.7e+308, Dy=-1.7e+308, IsMathDy=true, Ddy=-1.7e+308, IsMathDdy=true, Dddy=-1.7e+308, IsMathDddy=true)
  Curve (Type=Polynomial5)
    LeftBoundary (IsDefinedDdy=false, Ddy=0, IsMathDdy=true, IsDefinedDddy=false, Dddy=0, IsMathDddy=true)
    RightBoundary (IsDefinedDdy=false, Ddy=0, IsMathDdy=true, IsDefinedDddy=false, Dddy=0, IsMathDddy=true)
    Spline3 (IsContinuous4Derivative=false, IsDefinedSaddlePoint=false, IsDefinedLineAs2ndSegment=false, IsDefinedSlopeOfLine=false, SlopeOfLine=0, IsMathSlopeOfLine=true)
    Supremum (y=1.7e+308, Dy=1.7e+308, IsMathDy=true, Ddy=1.7e+308, IsMathDdy=true, Dddy=1.7e+308, IsMathDddy=true)
    Infimum (y=-1.7e+308, Dy=-1.7e+308, IsMathDy=true, Ddy=-1.7e+308, IsMathDdy=true, Dddy=-1.7e+308, IsMathDddy=true)
  Cam (LeftBoundaryIndex=0, RightBoundaryIndex=5)
    Supremum (y=1.7e+308, Dy=1.7e+308, IsMathDy=true, Ddy=1.7e+308, IsMathDdy=true, Dddy=1.7e+308, IsMathDddy=true)
    Infimum (y=-1.7e+308, Dy=-1.7e+308, IsMathDy=true, Ddy=-1.7e+308, IsMathDdy=true, Dddy=1.7e+308, IsMathDddy=true)
  ChartExtensions
```

### Program Logical/BootleFiller

#### Types.typ
```iecst
TYPE
	FillerEnum :
		( (*Every possible case*)
		INIT,
		WORK,
		ERROR
		);
END_TYPE
```

#### Variables.var
```iecst
(*case machine*)
VAR
	roleInfo : MpUserXMgrUIRoleInfoType;
	FillerTyp : FillerEnum;
END_VAR
(*digital inputs*)
VAR
	diConveyorHomingSwitch : BOOL := FALSE; (*Sensor detecting conveyor at homing position*)
	diNozzleHomingSwitch : BOOL; (*Sensor detecting nozzle at homing position*)
	diCartHomingSwitch : USINT; (*Sensor detecting cart at homing position*)
	diBottleDetection : BOOL := FALSE; (*Sensor detecting presence of a bottle*)
END_VAR
(*digital outputs*)
VAR
	doPumpRelay : BOOL; (*Output controlling the pump building pressure for liquid flow*)
	doValveRelay : BOOL; (*Output controlling the liquid valve opening*)
END_VAR
(*analog outputs*)
VAR
	aoPumpFlowSpeed : ARRAY[0..100] OF INT; (*Datapoint in percentage to the pump system about liquid flow speed in percent*)
END_VAR
```

#### Main.st
```iecst
PROGRAM _INIT
	(* Insert code here *)
	 FillerTyp:=INIT;
END_PROGRAM

PROGRAM _CYCLIC
	(* Insert code here *)
	CASE FillerTyp OF
		INIT:

		WORK:

		ERROR:

	END_CASE;

END_PROGRAM

PROGRAM _EXIT
	(* Insert code here *)

END_PROGRAM
```

### Program Logical/Package/test (IEC)

#### Main.st
```iecst
PROGRAM _INIT
	(* Insert code here *)
	FillerTyp:=DISABLED;
END_PROGRAM

PROGRAM _CYCLIC
	(* Insert code here *)
	MpBFRecipeXml(MpLink := ADR(BFRecipe) , Enable := 1, DeviceName := ADR('USER') , FileName := ADR('BottleFillerRecipe'));
	MpBFRecipeRegPar(MpLink := ADR(BFRecipe), Enable := 1, PVName := ADR('BootleFiller:bottleFillerRecipeTyp'));
	//MpBFRecipeHMI(MpLink := ADR(BFRecipe), Enable := 1 , ErrorReset := , UISetup := ADR(UISetup) , UIConnect := ADR(MpRecipeUIConnectType));

	MpBFRecipeXml();
	//MpBFRecipeHMI();
	CASE FillerTyp OF
		DISABLED:

		INIT:

		AUTOMAT:

		SERVICE:

		ERROR:

		STOP:

	END_CASE;

END_PROGRAM

PROGRAM _EXIT
	(* Insert code here *)

END_PROGRAM
```

### BF_GlobarVar.var
```iecst
VAR
	gFillerTyp : gBFWorkEnum;
	gAxisCase : gBFCaseEnum;
	gControl : gManagementTyp;
	gAxisUpdate : gAxisUpdateParType;
	gMainAction : gMainActionTyp;
	gAxisOutputs : gAxisOutputsTyp;
END_VAR
```

### BF_GlobalTyp.typ
```iecst
TYPE
	camSequencersParams : 	STRUCT
		cart : camParam;
		nozzle : camParam;
	END_STRUCT;
	camParam : 	STRUCT
		signal1 : BOOL := FALSE;
		currentStateIndex : INT := 0;
	END_STRUCT;
	gAxisOutputsTyp : 	STRUCT
		Conveyor : gControlInfoTyp;
		Cart : gControlInfoTyp;
		Nozzle : gControlInfoTyp;
		currentBottleType : UINT := 1;
	END_STRUCT;
	gControlInfoTyp : 	STRUCT  (*parameters, output*)
		error : BOOL := FALSE;
		isPowered : BOOL := FALSE;
		isHomed : BOOL := FALSE;
		position : REAL := 0;
		velocity : REAL := 0;
		updateDone : BOOL := FALSE;
		MoveActive : BOOL := FALSE;
	END_STRUCT;
	gControlTyp : 	STRUCT  (*parameters, inputs*)
		power : BOOL := FALSE;
		errorReset : BOOL := FALSE;
		home : BOOL := FALSE;
		jogNegative : BOOL := FALSE;
		jogPositive : BOOL := FALSE;
		moveVelocity : BOOL := FALSE;
		stop : BOOL := FALSE;
		currentBottleType : STRING[80] := '1';
		safeLevelStop : BOOL;
		onlyLeft : BOOL := FALSE;
		onlyRight : BOOL := FALSE;
		upperLimit : INT;
		lowerLimit : INT;
	END_STRUCT;
	gMainActionTyp : 	STRUCT
		powered : BOOL := FALSE;
		homed : BOOL := FALSE;
		connected : BOOL := FALSE;
		disconnected : BOOL := FALSE;
		stopped : BOOL := FALSE;
	END_STRUCT;
	gAxisUpdateParType : 	STRUCT  (*update parameters structure*)
		Conveyor : gParametersUpdate;
		Cart : gParametersUpdate;
		Nozzle : gParametersUpdate;
		staticVelocity : STRING[80] := '10';
	END_STRUCT;
	gManagementTyp : 	STRUCT
		Conveyor : gControlTyp;
		Cart : gControlTyp;
		Nozzle : gControlTyp;
		power : BOOL := FALSE;
		start : BOOL := FALSE;
		stop : BOOL := FALSE;
		manual : BOOL := FALSE;
		inCam : BOOL := FALSE;
		needUpdate : BOOL := FALSE;
		moveVelocity : BOOL := FALSE;
		disconnect : BOOL := FALSE;
		bottleCnt : INT := 0;
		currentBottleType : STRING[80] := '1';
	END_STRUCT;
	gParametersUpdate : 	STRUCT  (*update parameters*)
		Velocity : REAL := 10;
		Direction : REAL := 1;
		FirstPosition : REAL := 0;
		LastPosition : REAL := 0;
		Position : REAL := 0;
		Homing : REAL := 0;
	END_STRUCT;
	gBFWorkEnum :
		( (*BF_Work control*)
		WAITING,
		MANUAL,
		AUTOMAT
		);
	gBFCaseEnum :
		( (*BF_Axis control*)
		WAIT,
		POWERED,
		HOLDON,
		HOMING,
		CONNECT,
		STANDSTILL,
		onMOVE,
		DISCONNECT
		);
END_TYPE
```

### GlobalRobVis.var - Global variables
```iecst
VAR
	gAdrAxesPositions : UDINT;
	gMachineInterface : MachineAPIType;
END_VAR
```

### Program Logical/Simulation/Logic/RobVis (IEC)

#### Types.typ
```iecst
TYPE
	ModelConfigBottleType : 	STRUCT
		CenterToCenter : REAL; (*Bottle center to center in line*)
		Diameter : REAL; (*Bottle diameter*)
		Gap : REAL; (*Gap between bottles*)
	END_STRUCT;
	ModelConfigType : 	STRUCT
		Bottle : ModelConfigBottleType;
	END_STRUCT;
	RobVisPosType : 	STRUCT
		Conveyor : REAL;
		Cart : REAL;
		Nozzle : REAL;
		SensorColor : USINT;
	END_STRUCT;
END_TYPE
```

#### Variables.var
```iecst
VAR
	cmdTestModelMovements : BOOL;
	RobVisData : RobVisPosType;
	ModelConfig : ModelConfigType;
	i : INT;
	diBottleOld : BOOL;
	ConveyorAxisPosition : REAL;
	CartAxisPosition : REAL;
	NozzleAxisPosition : REAL;
	pAxesPositions : REFERENCE TO AxesPositionsType;
	AxesPosition : AxesPositionsType;
	bottleStartPoint : REAL;
	bottleEndPoint : REAL;
	diBottle: BOOL := FALSE;
	cntBottle : UDINT := 0;
END_VAR
```

#### Main.st
```iecst
PROGRAM _INIT

	ModelConfig.Bottle.CenterToCenter := 100;
	ModelConfig.Bottle.Diameter := 80;
	ModelConfig.Bottle.Gap := ModelConfig.Bottle.CenterToCenter - ModelConfig.Bottle.Diameter;

	RobVisData.Conveyor := 0.0;
	RobVisData.Cart := 0.0;
	RobVisData.Nozzle := 195.0;
END_PROGRAM

PROGRAM _CYCLIC

	//gAdrAxesPositions := ADR(AxesPosition);

	IF gAdrAxesPositions <> 0 THEN
		pAxesPositions ACCESS gAdrAxesPositions;
	ELSE
		RETURN;
	END_IF

	// --------------------------------------------
	// Prepare correct positions for model
	// --------------------------------------------
	RobVisData.Conveyor := LREAL_TO_REAL(pAxesPositions.Conveyor + ConveyorAxisPosition);
	RobVisData.Cart := LREAL_TO_REAL(pAxesPositions.Cart + CartAxisPosition);
	RobVisData.Nozzle := LREAL_TO_REAL(pAxesPositions.Nozzle + NozzleAxisPosition);
	RobVisData.SensorColor;

	// Homing Switches Control
	gMachineInterface.DigitalInputs.ConveyorHomingSwitch := diBottle AND (cntBottle MOD 5 = 1);
	gMachineInterface.DigitalInputs.CartHomingSwitch := RobVisData.Cart <= -50;
	gMachineInterface.DigitalInputs.NozzleHomingSwitch := RobVisData.Nozzle >= 195;

	// --------------------------------------------
	// Bottle Signal Generator
	// --------------------------------------------
	FOR i := 0 TO 50 DO
		bottleStartPoint := i*ModelConfig.Bottle.CenterToCenter + ModelConfig.Bottle.Diameter + ModelConfig.Bottle.Gap/2;
		bottleEndPoint := bottleStartPoint + ModelConfig.Bottle.Diameter;

		IF (RobVisData.Conveyor > bottleStartPoint) AND (RobVisData.Conveyor < bottleEndPoint) THEN
			diBottle := TRUE;
			RobVisData.SensorColor := 5;
			EXIT;
		ELSE
			diBottle := FALSE;
			RobVisData.SensorColor := 11;
		END_IF
	END_FOR

	// --------------------------------------------
	// Bottle counter
	// --------------------------------------------
	IF (diBottleOld <> diBottle) AND diBottle THEN
		cntBottle := cntBottle + 1;
		gControl.bottleCnt:= gControl.bottleCnt + 1;
	END_IF
	diBottleOld := diBottle;

	// --------------------------------------------
	// Tests
	// --------------------------------------------
	IF cmdTestModelMovements THEN
		ConveyorAxisPosition := ConveyorAxisPosition + 1;
		CartAxisPosition := CartAxisPosition + 1;
		NozzleAxisPosition := NozzleAxisPosition + 1;

		IF ConveyorAxisPosition > 2500 THEN
			ConveyorAxisPosition := 0;
		END_IF

		IF CartAxisPosition > 1200 THEN
			CartAxisPosition := 0;
		END_IF

		IF NozzleAxisPosition > 200 THEN
			NozzleAxisPosition := 0;
		END_IF
	END_IF

END_PROGRAM
```

### Program Logical/Simulation/Logic/BF_Main (IEC)

#### Variables.var
```iecst
(*case machine*)
VAR
	FillerTyp : FillerEnum;
	bottleFillerRecipeTyp : bottleFillerRecipeEnum;
END_VAR
(*digital inputs*)
VAR
	diError : BOOL;
	diManual : BOOL := FALSE; (*Determine if machine works automatically or needs manual control*)
	diStop : BOOL := FALSE; (*Stop switch*)
	diStart : BOOL := FALSE; (*Start switch*)
	diPowerSwitch : BOOL := FALSE; (*Power on switch*)
	diLiquidLevel : REAL := 100;
	diConveyorHomingSwitch : BOOL := FALSE; (*Sensor detecting conveyor at homing position*)
	diNozzleHomingSwitch : BOOL := FALSE; (*Sensor detecting nozzle at homing position*)
	diCartHomingSwitch : BOOL := FALSE; (*Sensor detecting cart at homing position*)
	diBottleDetection : BOOL := FALSE; (*Sensor detecting presence of a bottle*)
END_VAR
(*digital outputs*)
VAR
	doPumpRelay : INT; (*Output controlling the pump building pressure for liquid flow*)
	doValveRelay : BOOL; (*Output controlling the liquid valve opening*)
END_VAR
(*analog outputs*)
VAR
	aoPumpFlowSpeed : ARRAY[0..100] OF INT; (*Datapoint in percentage to the pump system about liquid flow speed in percent*)
END_VAR
(*other variables*)
VAR
	result : INT;
	counter : INT;
	roleInfo : MpUserXMgrUIRoleInfoType;
	MpBFRecipeXml : MpRecipeXml;
	MpBFRecipeRegPar : MpRecipeRegPar; (*MpBFRecipeHMI : MpRecipeUI;
	UISetup : MpRecipeUISetupType;
	MpRecipeUIConnectType : MpRecipeUIConnectType;*)
	inCam : BOOL;
	SimulationAxisPosition : SimulationAxisPositionEnum;
	changedPosition : BOOL;
END_VAR
```

#### Main.st
```iecst
PROGRAM _INIT
	(* Insert code here *)
	 FillerTyp:=DISABLED;
END_PROGRAM

PROGRAM _CYCLIC
	(* Insert code here *)

	SimulationAxisPosition.Cart := LREAL_TO_REAL(gAxisOutputs.Cart.position);
	SimulationAxisPosition.Conveyor := LREAL_TO_REAL(gAxisOutputs.Conveyor.position);
	SimulationAxisPosition.Nozzle := LREAL_TO_REAL(gAxisOutputs.Nozzle.position);
	gAdrAxesPositions := ADR(SimulationAxisPosition);

	CASE FillerTyp OF
		DISABLED:
			diStart:=0;
			diStop:=0;

			IF gControl.power THEN
				FillerTyp:=INIT;
			END_IF;

		INIT:
			gControl.Cart.lowerLimit:=-95;
			gControl.Cart.upperLimit:=1095;

			gControl.Conveyor.lowerLimit:=0;
			gControl.Conveyor.upperLimit:=4997;

			gControl.Nozzle.lowerLimit:=2;
			gControl.Nozzle.upperLimit:=197;

			gAxisCase:=POWERED;

			IF gMainAction.powered THEN
				gAxisCase:=HOMING;
			END_IF;

			IF gMainAction.powered AND gMainAction.homed THEN
				gControl.Cart.home:=0;
				gControl.Conveyor.home:=0;
				gControl.Nozzle.home:=0;
				gAxisCase:=STANDSTILL;
			END_IF;

			IF gMainAction.powered AND gMainAction.homed AND gControl.start AND NOT gControl.manual THEN
				gAxisCase:=CONNECT;
				IF gMainAction.connected THEN
					gAxisCase:=onMOVE;
					gFillerTyp:=AUTOMAT;
					FillerTyp:=WORK;
				END_IF;
			END_IF;

			IF gMainAction.powered AND gMainAction.homed AND gControl.start AND gControl.manual THEN
				gMainAction.homed:=0;
				gAxisCase:=onMOVE;
				gFillerTyp:=MANUAL;
				FillerTyp:=WORK;
			END_IF;

		WORK:
			result:= gControl.bottleCnt MOD 5;

			IF result=1 THEN
				gCamSeqParam.nozzle.signal1:=1;
			END_IF;
			IF result <> 1 THEN
				gCamSeqParam.nozzle.signal1:=0;
				gCamSeqParam.cart.signal1:=0;
			END_IF;

		ERROR:

		STOP:

	END_CASE;

END_PROGRAM

PROGRAM _EXIT
	(* Insert code here *)

END_PROGRAM
```

### Program Logical/Simulation/Logic/BF_Work (IEC)

#### Types.typ
```iecst
TYPE
	controlTyp :
		(
		HOMING,
		ERROR,
		MANUAL,
		STOP,
		AUTOMATIC,
		INIT
		);
END_TYPE
```

#### Variables.var
```iecst
VAR
	fillerTyp : controlTyp;
END_VAR
```

#### Main.st
```iecst
PROGRAM _INIT
	(* Insert code here *)
END_PROGRAM

PROGRAM _CYCLIC
	(* Insert code here *)

	CASE gFillerTyp OF

		MANUAL:

			IF EDGENEG(gAxisOutputs.Cart.MoveActive) THEN
				gControl.Cart.jogNegative:=0;
				gControl.Cart.jogPositive:=0;
			END_IF;

			IF EDGENEG(gAxisOutputs.Conveyor.MoveActive) THEN
				gControl.Conveyor.jogNegative:=0;
				gControl.Conveyor.jogPositive:=0;
			END_IF;
			IF 	EDGENEG(gAxisOutputs.Nozzle.MoveActive) THEN
				gControl.Nozzle.jogNegative:=0;
				gControl.Nozzle.jogPositive:=0;
			END_IF;

			IF EDGEPOS(gControl.inCam) THEN
				switch:=1;
			END_IF;

			IF EDGENEG(gControl.inCam) THEN
				switch:=2;
			END_IF;

			IF switch=1 OR EDGEPOS(gControl.inCam) THEN
				IF NOT gMainAction.stopped THEN
					gAxisCase:=HOLDON;
				END_IF;

				IF gMainAction.stopped AND NOT gMainAction.homed THEN
					gAxisCase:=HOMING;
				END_IF;

				IF gMainAction.stopped AND gMainAction.homed AND NOT gMainAction.connected THEN
					gMainAction.disconnected:=0;
					gAxisCase:=CONNECT;
				END_IF;

				IF gMainAction.stopped AND gMainAction.connected AND gMainAction.homed THEN
					gControl.Cart.home:=0;
					gControl.Conveyor.home:=0;
					gControl.Nozzle.home:=0;
					gMainAction.homed:=0;

					gMainAction.stopped:=0;
					gAxisCase:=onMOVE;
					switch:=0;
				END_IF;
			END_IF;

			IF switch=2 OR EDGENEG(gControl.inCam) THEN
				IF NOT gMainAction.disconnected THEN
					gAxisCase:=DISCONNECT;
					gMainAction.connected:=0;
				END_IF;

				IF gMainAction.disconnected THEN
					gControl.Cart.home:=0;
					gControl.Conveyor.home:=0;
					gControl.Nozzle.home:=0;
					gMainAction.homed:=0;
					gAxisCase:=onMOVE;
					IF gAxisCase=onMOVE THEN
						switch:=0;
					END_IF;
				END_IF;
			END_IF;

			IF NOT gControl.manual THEN
				gAxisCase:=HOMING;
				IF gMainAction.homed THEN
					gControl.Cart.home:=0;
					gControl.Conveyor.home:=0;
					gControl.Nozzle.home:=0;
					gAxisCase:=CONNECT;
					gMainAction.disconnected:=0;
					IF gMainAction.connected THEN
						gMainAction.homed:=0;
						switch:=0;
						gFillerTyp:=AUTOMAT;
						gAxisCase:=onMOVE;
					END_IF;
				END_IF;
			END_IF;

			//zabezpieczenia przed przejechaniem manualnym poza limit
			IF gAxisOutputs.Cart.position <= gControl.Cart.lowerLimit OR gAxisOutputs.Cart.position >= gControl.Cart.upperLimit THEN
				gControl.Cart.safeLevelStop:=1;
				IF gAxisOutputs.Cart.position >= gControl.Cart.upperLimit THEN
					gControl.Cart.onlyLeft:=1;
				ELSE
					gControl.Cart.onlyRight:=1;
				END_IF;
			ELSE
				gControl.Cart.onlyLeft:=0;
				gControl.Cart.onlyRight:=0;
				gControl.Cart.safeLevelStop:=0;
			END_IF;

			IF gAxisOutputs.Nozzle.position <= gControl.Nozzle.lowerLimit OR gAxisOutputs.Nozzle.position >= gControl.Nozzle.upperLimit THEN
				gControl.Nozzle.safeLevelStop:=1;
				IF gAxisOutputs.Nozzle.position <= gControl.Nozzle.lowerLimit THEN
					gControl.Nozzle.onlyRight:=1;
				ELSE
					gControl.Nozzle.onlyLeft:=1;
				END_IF;
			ELSE
				gControl.Nozzle.safeLevelStop:=0;
				gControl.Nozzle.onlyLeft:=0;
				gControl.Nozzle.onlyRight:=0;
			END_IF;

		AUTOMAT:

			gControl.moveVelocity:= gControl.start AND (NOT gControl.stop);
			IF gControl.manual THEN
				gControl.moveVelocity:=0;
				gAxisCase:=DISCONNECT;
				IF gMainAction.disconnected THEN
					gFillerTyp:=MANUAL;
				END_IF;
			END_IF;

	END_CASE;

END_PROGRAM

PROGRAM _EXIT
	(* Insert code here *)

END_PROGRAM
```

### Program Logical/Simulation/Logic/BF_Axis (IEC)

#### Types.typ
```iecst
TYPE
	axisCaseEnum :
		(
		POWERED,
		HOMING,
		onMOVE,
		CONNECT,
		STANDSTILL,
		UPDATE
		);
	managementTyp : 	STRUCT
		Conveyor : manualControlTyp;
		Cart : manualControlTyp;
		Nozzle : manualControlTyp;
	END_STRUCT;
	InfosTyp : 	STRUCT
		Conveyor : manualControlInfoTyp;
		Cart : manualControlInfoTyp;
		Nozzle : manualControlInfoTyp;
	END_STRUCT;
	manualControlInfoTyp : 	STRUCT
		error : BOOL;
		isPowered : BOOL;
		isHomed : BOOL;
	END_STRUCT;
	manualControlTyp : 	STRUCT
		errorReset : BOOL;
		start : BOOL;
		home : BOOL;
		jogNegative : BOOL;
		jogPositive : BOOL;
		stop : BOOL;
	END_STRUCT;
	axisesManagementType : 	STRUCT
		diStart : BOOL;
		diError : BOOL;
		diManual : BOOL;
		diPowerSwitch : BOOL;
		diStop : BOOL;
	END_STRUCT;
END_TYPE
```

#### Variables.var
```iecst
(*Axises*)
VAR
	MpAxisConv : MpAxisBasic;
	MpAxisCart : MpAxisBasic;
	MpAxisNozzle : MpAxisBasic;
END_VAR
(*Axis Parameters*)
VAR
	MpAxisCartParType : MpAxisBasicParType;
	MpAxisNozzleParType : MpAxisBasicParType;
	MpAxisConvParType : MpAxisBasicParType;
END_VAR
(*Cam Variables*)
VAR
	camSeq : MpAxisCamSequencer;
	camSeqNozzle : MpAxisCamSequencer;
	camNozzleParameters : MpAxisCamSequencerParType;
	configCamNozzle : McAcpAxCamAutParType;
	camParameters : MpAxisCamSequencerParType;
END_VAR
(*Other Variables*)
VAR
	needUpdate : BOOL := FALSE;
	homed : BOOL := FALSE; (*defines if all the axises are homed*)
END_VAR
(*global used variables*)
VAR
	axisMgmt : axisesManagementType;
	controlInfo : gAxisOutputsTyp;
	connectHelper : INT := 0;
	handleStopCart : BOOL := FALSE;
	handleStopNozzle : BOOL := FALSE;
END_VAR
```
